LIN {X 0,Y 531.026,Z 365.335,A -85,B 0,C 180,E1 -4215.435,E2 -4215.435} C_VEL
LIN {X 0,Y 531.043,Z 365.34,A -85,B 0,C 180,E1 -4218.549,E2 -4218.549} C_VEL
LIN {X 0,Y 531.061,Z 365.329,A -85,B 0,C 180,E1 -4221.629,E2 -4221.629} C_VEL
LIN {X 0,Y 531.122,Z 365.326,A -85,B 0,C 180,E1 -4224.684,E2 -4224.684} C_VEL
LIN {X 0,Y 531.145,Z 365.319,A -85,B 0,C 180,E1 -4227.724,E2 -4227.724} C_VEL
LIN {X 0,Y 531.157,Z 365.319,A -85,B 0,C 180,E1 -4230.757,E2 -4230.757} C_VEL
LIN {X 0,Y 531.108,Z 365.323,A -85,B 0,C 180,E1 -4233.033,E2 -4233.033} C_VEL
LIN {X 0,Y 531.087,Z 365.332,A -85,B 0,C 180,E1 -4236.076,E2 -4236.076} C_VEL
LIN {X 0,Y 531.056,Z 365.335,A -85,B 0,C 180,E1 -4238.369,E2 -4238.369} C_VEL
LIN {X 0,Y 531.054,Z 365.332,A -85,B 0,C 180,E1 -4241.671,E2 -4241.671} C_VEL
LIN {X 0,Y 531.033,Z 365.332,A -85,B 0,C 180,E1 -4244.955,E2 -4244.955} C_VEL
LIN {X 0,Y 531.018,Z 365.339,A -85,B 0,C 180,E1 -4247.721,E2 -4247.721} C_VEL
LIN {X 0,Y 531.025,Z 365.339,A -85,B 0,C 180,E1 -4250.126,E2 -4250.126} C_VEL
LIN {X 0,Y 530.946,Z 365.344,A -85,B 0,C 180,E1 -4252.572,E2 -4252.572} C_VEL
LIN {X 0,Y 530.994,Z 365.337,A -85,B 0,C 180,E1 -4255.057,E2 -4255.057} C_VEL
LIN {X 0,Y 531.015,Z 365.34,A -85,B 0,C 180,E1 -4257.594,E2 -4257.594} C_VEL
LIN {X 0,Y 530.981,Z 365.339,A -85,B 0,C 180,E1 -4260.646,E2 -4260.646} C_VEL
LIN {X 0,Y 530.988,Z 365.346,A -85,B 0,C 180,E1 -4263.771,E2 -4263.771} C_VEL
LIN {X 0,Y 530.965,Z 365.34,A -85,B 0,C 180,E1 -4266.556,E2 -4266.556} C_VEL
LIN {X 0,Y 530.996,Z 365.341,A -85,B 0,C 180,E1 -4269.855,E2 -4269.855} C_VEL
LIN {X 0,Y 530.978,Z 365.339,A -85,B 0,C 180,E1 -4272.455,E2 -4272.455} C_VEL
LIN {X 0,Y 530.983,Z 365.347,A -85,B 0,C 180,E1 -4275.62,E2 -4275.62} C_VEL
LIN {X 0,Y 531.042,Z 365.474,A -85,B 0,C 180,E1 -4277.77,E2 -4277.77} C_VEL
LIN {X 0,Y 531.558,Z 369.985,A -85,B 0,C 180,E1 -4278.618,E2 -4278.618} C_VEL
LIN {X 0,Y 531.348,Z 387.405,A -85,B 0,C 180,E1 -4281.804,E2 -4281.804} C_VEL
LIN {X 0,Y 531.197,Z 394.529,A -85,B 0,C 180,E1 -4283.118,E2 -4283.118} C_VEL
LIN {X 0,Y 532.782,Z 405.07,A -85,B 0,C 180,E1 -4283.315,E2 -4283.315} C_VEL
LIN {X 0,Y 532.355,Z 500.213,A -85,B 0,C 180,E1 -4284.624,E2 -4284.624} C_VEL
LIN {X 0,Y 532.243,Z 511.094,A -85,B 0,C 180,E1 -4284.875,E2 -4284.875} C_VEL
LIN {X 0,Y 532.076,Z 522.958,A -85,B 0,C 180,E1 -4285.275,E2 -4285.275} C_VEL
LIN {X 0,Y 531.831,Z 535.01,A -85,B 0,C 180,E1 -4285.831,E2 -4285.831} C_VEL
LIN {X 0,Y 531.61,Z 545.985,A -85,B 0,C 180,E1 -4286.499,E2 -4286.499} C_VEL
LIN {X 0,Y 531.342,Z 555.982,A -85,B 0,C 180,E1 -4287.257,E2 -4287.257} C_VEL
LIN {X 0,Y 531.14,Z 564.562,A -85,B 0,C 180,E1 -4288.043,E2 -4288.043} C_VEL
LIN {X 0,Y 530.97,Z 572.57,A -85,B 0,C 180,E1 -4288.921,E2 -4288.921} C_VEL
LIN {X 0,Y 530.813,Z 579.244,A -85,B 0,C 180,E1 -4289.793,E2 -4289.793} C_VEL
LIN {X 0,Y 530.664,Z 584.849,A -85,B 0,C 180,E1 -4290.658,E2 -4290.658} C_VEL
LIN {X 0,Y 530.582,Z 590.653,A -85,B 0,C 180,E1 -4291.736,E2 -4291.736} C_VEL
LIN {X 0,Y 530.512,Z 595.671,A -85,B 0,C 180,E1 -4292.899,E2 -4292.899} C_VEL
LIN {X 0,Y 530.466,Z 600.121,A -85,B 0,C 180,E1 -4294.275,E2 -4294.275} C_VEL
LIN {X 0,Y 530.387,Z 603.167,A -85,B 0,C 180,E1 -4295.746,E2 -4295.746} C_VEL
LIN {X 0,Y 530.394,Z 604.282,A -85,B 0,C 180,E1 -4296.577,E2 -4296.577} C_VEL
LIN {X 0,Y 530.349,Z 604.907,A -85,B 0,C 180,E1 -4297.4,E2 -4297.4} C_VEL
LIN {X 0,Y 530.396,Z 604.976,A -85,B 0,C 180,E1 -4298.222,E2 -4298.222} C_VEL
LIN {X 0,Y 530.35,Z 603.932,A -85,B 0,C 180,E1 -4299.846,E2 -4299.846} C_VEL
LIN {X 0,Y 530.381,Z 602.696,A -85,B 0,C 180,E1 -4300.654,E2 -4300.654} C_VEL
LIN {X 0,Y 530.464,Z 600.013,A -85,B 0,C 180,E1 -4301.859,E2 -4301.859} C_VEL
LIN {X 0,Y 530.485,Z 596.223,A -85,B 0,C 180,E1 -4303.054,E2 -4303.054} C_VEL
LIN {X 0,Y 530.552,Z 591.215,A -85,B 0,C 180,E1 -4304.243,E2 -4304.243} C_VEL
LIN {X 0,Y 530.673,Z 586.337,A -85,B 0,C 180,E1 -4305.185,E2 -4305.185} C_VEL
LIN {X 0,Y 530.795,Z 579.863,A -85,B 0,C 180,E1 -4306.212,E2 -4306.212} C_VEL
LIN {X 0,Y 530.963,Z 572.403,A -85,B 0,C 180,E1 -4307.19,E2 -4307.19} C_VEL
LIN {X 0,Y 531.141,Z 564.201,A -85,B 0,C 180,E1 -4308.085,E2 -4308.085} C_VEL
LIN {X 0,Y 531.385,Z 554.7,A -85,B 0,C 180,E1 -4308.944,E2 -4308.944} C_VEL
LIN {X 0,Y 531.696,Z 542.537,A -85,B 0,C 180,E1 -4309.817,E2 -4309.817} C_VEL
LIN {X 0,Y 531.902,Z 531.205,A -85,B 0,C 180,E1 -4310.445,E2 -4310.445} C_VEL
LIN {X 0,Y 532.087,Z 519.921,A -85,B 0,C 180,E1 -4310.928,E2 -4310.928} C_VEL
LIN {X 0,Y 532.288,Z 507.418,A -85,B 0,C 180,E1 -4311.314,E2 -4311.314} C_VEL
LIN {X 0,Y 532.422,Z 491.23,A -85,B 0,C 180,E1 -4311.603,E2 -4311.603} C_VEL
LIN {X 0,Y 532.675,Z 403.02,A -85,B 0,C 180,E1 -4312.807,E2 -4312.807} C_VEL
LIN {X 0,Y 531.213,Z 394.5,A -85,B 0,C 180,E1 -4312.992,E2 -4312.992} C_VEL
LIN {X 0,Y 531.363,Z 379.959,A -85,B 0,C 180,E1 -4315.638,E2 -4315.638} C_VEL
LIN {X 0,Y 531.455,Z 369.437,A -85,B 0,C 180,E1 -4317.537,E2 -4317.537} C_VEL
LIN {X 0,Y 531.071,Z 365.336,A -85,B 0,C 180,E1 -4318.294,E2 -4318.294} C_VEL
LIN {X 0,Y 531.147,Z 365.326,A -85,B 0,C 180,E1 -4320.758,E2 -4320.758} C_VEL
LIN {X 0,Y 531.101,Z 365.329,A -85,B 0,C 180,E1 -4323.034,E2 -4323.034} C_VEL
LIN {X 0,Y 531.075,Z 365.333,A -85,B 0,C 180,E1 -4326.077,E2 -4326.077} C_VEL
LIN {X 0,Y 531.027,Z 365.335,A -85,B 0,C 180,E1 -4329.138,E2 -4329.138} C_VEL
LIN {X 0,Y 531.031,Z 365.34,A -85,B 0,C 180,E1 -4332.225,E2 -4332.225} C_VEL
LIN {X 0,Y 530.987,Z 365.34,A -85,B 0,C 180,E1 -4335.35,E2 -4335.35} C_VEL
LIN {X 0,Y 531.006,Z 365.341,A -85,B 0,C 180,E1 -4337.723,E2 -4337.723} C_VEL
LIN {X 0,Y 530.998,Z 365.337,A -85,B 0,C 180,E1 -4340.938,E2 -4340.938} C_VEL
LIN {X 0,Y 531.018,Z 365.341,A -85,B 0,C 180,E1 -4344.05,E2 -4344.05} C_VEL
LIN {X 0,Y 531.006,Z 365.336,A -85,B 0,C 180,E1 -4346.744,E2 -4346.744} C_VEL
LIN {X 0,Y 530.991,Z 365.342,A -85,B 0,C 180,E1 -4349.322,E2 -4349.322} C_VEL
LIN {X 0,Y 530.972,Z 365.343,A -85,B 0,C 180,E1 -4352.104,E2 -4352.104} C_VEL
LIN {X 0,Y 530.983,Z 365.34,A -85,B 0,C 180,E1 -4354.855,E2 -4354.855} C_VEL
LIN {X 0,Y 530.959,Z 365.35,A -85,B 0,C 180,E1 -4357.508,E2 -4357.508} C_VEL
LIN {X 0,Y 530.978,Z 365.34,A -85,B 0,C 180,E1 -4360.433,E2 -4360.433} C_VEL
LIN {X 0,Y 530.961,Z 365.347,A -85,B 0,C 180,E1 -4363.495,E2 -4363.495} C_VEL
LIN {X 0,Y 530.958,Z 365.343,A -85,B 0,C 180,E1 -4366.507,E2 -4366.507} C_VEL
LIN {X 0,Y 530.984,Z 365.346,A -85,B 0,C 180,E1 -4368.977,E2 -4368.977} C_VEL
LIN {X 0,Y 530.955,Z 365.345,A -85,B 0,C 180,E1 -4371.531,E2 -4371.531} C_VEL
LIN {X 0,Y 530.979,Z 365.341,A -85,B 0,C 180,E1 -4374.383,E2 -4374.383} C_VEL
LIN {X 0,Y 530.969,Z 365.346,A -85,B 0,C 180,E1 -4377.135,E2 -4377.135} C_VEL
LIN {X 0,Y 530.984,Z 365.34,A -85,B 0,C 180,E1 -4379.805,E2 -4379.805} C_VEL
LIN {X 0,Y 531.016,Z 365.341,A -85,B 0,C 180,E1 -4382.467,E2 -4382.467} C_VEL
LIN {X 0,Y 531.007,Z 365.344,A -85,B 0,C 180,E1 -4384.944,E2 -4384.944} C_VEL
LIN {X 0,Y 531.039,Z 365.539,A -85,B 0,C 180,E1 -4386.001,E2 -4386.001} C_VEL
LIN {X 0,Y 532.353,Z 373.078,A -85,B 0,C 180,E1 -4387.286,E2 -4387.286} C_VEL
LIN {X 0,Y 531.956,Z 390.881,A -85,B 0,C 180,E1 -4390.112,E2 -4390.112} C_VEL
LIN {X 0,Y 531.575,Z 408.654,A -85,B 0,C 180,E1 -4392.893,E2 -4392.893} C_VEL
LIN {X 0,Y 531.338,Z 422.569,A -85,B 0,C 180,E1 -4395.054,E2 -4395.054} C_VEL
LIN {X 0,Y 532.834,Z 432.971,A -85,B 0,C 180,E1 -4395.239,E2 -4395.239} C_VEL
LIN {X 0,Y 532.412,Z 530.394,A -85,B 0,C 180,E1 -4396.572,E2 -4396.572} C_VEL
LIN {X 0,Y 532.216,Z 543.761,A -85,B 0,C 180,E1 -4396.907,E2 -4396.907} C_VEL
LIN {X 0,Y 531.997,Z 555.976,A -85,B 0,C 180,E1 -4397.363,E2 -4397.363} C_VEL
LIN {X 0,Y 531.74,Z 568.122,A -85,B 0,C 180,E1 -4397.976,E2 -4397.976} C_VEL
LIN {X 0,Y 531.507,Z 579.917,A -85,B 0,C 180,E1 -4398.754,E2 -4398.754} C_VEL
LIN {X 0,Y 531.219,Z 590.378,A -85,B 0,C 180,E1 -4399.616,E2 -4399.616} C_VEL
LIN {X 0,Y 531.032,Z 598.931,A -85,B 0,C 180,E1 -4400.479,E2 -4400.479} C_VEL
LIN {X 0,Y 530.885,Z 606.821,A -85,B 0,C 180,E1 -4401.436,E2 -4401.436} C_VEL
LIN {X 0,Y 530.68,Z 614.522,A -85,B 0,C 180,E1 -4402.582,E2 -4402.582} C_VEL
LIN {X 0,Y 530.604,Z 621.622,A -85,B 0,C 180,E1 -4403.918,E2 -4403.918} C_VEL
LIN {X 0,Y 530.459,Z 626.341,A -85,B 0,C 180,E1 -4405.061,E2 -4405.061} C_VEL
LIN {X 0,Y 530.516,Z 629.95,A -85,B 0,C 180,E1 -4406.203,E2 -4406.203} C_VEL
LIN {X 0,Y 530.457,Z 631.806,A -85,B 0,C 180,E1 -4406.963,E2 -4406.963} C_VEL
LIN {X 0,Y 530.41,Z 633.194,A -85,B 0,C 180,E1 -4407.723,E2 -4407.723} C_VEL
LIN {X 0,Y 530.344,Z 634.786,A -85,B 0,C 180,E1 -4409.242,E2 -4409.242} C_VEL
LIN {X 0,Y 530.342,Z 635,A -85,B 0,C 180,E1 -4410.001,E2 -4410.001} C_VEL
LIN {X 0,Y 530.361,Z 634.182,A -85,B 0,C 180,E1 -4411.52,E2 -4411.52} C_VEL
LIN {X 0,Y 530.411,Z 633.194,A -85,B 0,C 180,E1 -4412.279,E2 -4412.279} C_VEL
LIN {X 0,Y 530.457,Z 631.805,A -85,B 0,C 180,E1 -4413.039,E2 -4413.039} C_VEL
LIN {X 0,Y 530.523,Z 628.874,A -85,B 0,C 180,E1 -4414.179,E2 -4414.179} C_VEL
LIN {X 0,Y 530.525,Z 624.9,A -85,B 0,C 180,E1 -4415.322,E2 -4415.322} C_VEL
LIN {X 0,Y 530.6,Z 619.178,A -85,B 0,C 180,E1 -4416.583,E2 -4416.583} C_VEL
LIN {X 0,Y 530.737,Z 612.104,A -85,B 0,C 180,E1 -4417.802,E2 -4417.802} C_VEL
LIN {X 0,Y 530.929,Z 603.811,A -85,B 0,C 180,E1 -4418.949,E2 -4418.949} C_VEL
LIN {X 0,Y 531.123,Z 595.305,A -85,B 0,C 180,E1 -4419.906,E2 -4419.906} C_VEL
LIN {X 0,Y 531.379,Z 584.793,A -85,B 0,C 180,E1 -4420.864,E2 -4420.864} C_VEL
LIN {X 0,Y 531.632,Z 573.998,A -85,B 0,C 180,E1 -4421.658,E2 -4421.658} C_VEL
LIN {X 0,Y 531.895,Z 562.981,A -85,B 0,C 180,E1 -4422.303,E2 -4422.303} C_VEL
LIN {X 0,Y 532.107,Z 551.244,A -85,B 0,C 180,E1 -4422.831,E2 -4422.831} C_VEL
LIN {X 0,Y 532.277,Z 538.628,A -85,B 0,C 180,E1 -4423.239,E2 -4423.239} C_VEL
LIN {X 0,Y 532.477,Z 525.779,A -85,B 0,C 180,E1 -4423.501,E2 -4423.501} C_VEL
LIN {X 0,Y 532.689,Z 431.415,A -85,B 0,C 180,E1 -4424.784,E2 -4424.784} C_VEL
LIN {X 0,Y 531.306,Z 422.381,A -85,B 0,C 180,E1 -4424.964,E2 -4424.964} C_VEL
LIN {X 0,Y 531.733,Z 402.026,A -85,B 0,C 180,E1 -4428.119,E2 -4428.119} C_VEL
LIN {X 0,Y 532.124,Z 381.772,A -85,B 0,C 180,E1 -4431.298,E2 -4431.298} C_VEL
LIN {X 0,Y 532.319,Z 372.885,A -85,B 0,C 180,E1 -4432.718,E2 -4432.718} C_VEL
LIN {X 0,Y 531.008,Z 365.342,A -85,B 0,C 180,E1 -4434.032,E2 -4434.032} C_VEL
LIN {X 0,Y 531.01,Z 365.339,A -85,B 0,C 180,E1 -4436.744,E2 -4436.744} C_VEL
LIN {X 0,Y 530.988,Z 365.348,A -85,B 0,C 180,E1 -4439.323,E2 -4439.323} C_VEL
LIN {X 0,Y 530.972,Z 365.342,A -85,B 0,C 180,E1 -4442.101,E2 -4442.101} C_VEL
LIN {X 0,Y 530.986,Z 365.343,A -85,B 0,C 180,E1 -4444.853,E2 -4444.853} C_VEL
LIN {X 0,Y 530.972,Z 365.346,A -85,B 0,C 180,E1 -4447.508,E2 -4447.508} C_VEL
LIN {X 0,Y 530.987,Z 365.341,A -85,B 0,C 180,E1 -4450.433,E2 -4450.433} C_VEL
LIN {X 0,Y 530.971,Z 365.344,A -85,B 0,C 180,E1 -4453.495,E2 -4453.495} C_VEL
LIN {X 0,Y 530.971,Z 365.344,A -85,B 0,C 180,E1 -4456.506,E2 -4456.506} C_VEL
LIN {X 0,Y 530.986,Z 365.338,A -85,B 0,C 180,E1 -4459.567,E2 -4459.567} C_VEL
LIN {X 0,Y 530.973,Z 365.345,A -85,B 0,C 180,E1 -4462.577,E2 -4462.577} C_VEL
LIN {X 0,Y 530.987,Z 365.339,A -85,B 0,C 180,E1 -4465.31,E2 -4465.31} C_VEL
LIN {X 0,Y 530.972,Z 365.341,A -85,B 0,C 180,E1 -4468.032,E2 -4468.032} C_VEL
LIN {X 0,Y 530.994,Z 365.343,A -85,B 0,C 180,E1 -4470.875,E2 -4470.875} C_VEL
LIN {X 0,Y 531.003,Z 365.335,A -85,B 0,C 180,E1 -4473.256,E2 -4473.256} C_VEL
LIN {X 0,Y 530.965,Z 365.343,A -85,B 0,C 180,E1 -4475.967,E2 -4475.967} C_VEL
LIN {X 0,Y 531.005,Z 365.338,A -85,B 0,C 180,E1 -4479.062,E2 -4479.062} C_VEL
LIN {X 0,Y 531.022,Z 365.338,A -85,B 0,C 180,E1 -4482.278,E2 -4482.278} C_VEL
LIN {X 0,Y 531.025,Z 365.331,A -85,B 0,C 180,E1 -4485.436,E2 -4485.436} C_VEL
LIN {X 0,Y 531.043,Z 365.335,A -85,B 0,C 180,E1 -4488.55,E2 -4488.55} C_VEL
LIN {X 0,Y 531.06,Z 365.331,A -85,B 0,C 180,E1 -4491.63,E2 -4491.63} C_VEL
LIN {X 0,Y 531.126,Z 365.323,A -85,B 0,C 180,E1 -4494.685,E2 -4494.685} C_VEL
LIN {X 0,Y 531.145,Z 365.32,A -85,B 0,C 180,E1 -4497.725,E2 -4497.725} C_VEL
LIN {X 0,Y 531.158,Z 365.317,A -85,B 0,C 180,E1 -4500.758,E2 -4500.758} C_VEL
LIN {X 0,Y 531.11,Z 365.323,A -85,B 0,C 180,E1 -4503.034,E2 -4503.034} C_VEL
LIN {X 0,Y 531.09,Z 365.332,A -85,B 0,C 180,E1 -4506.077,E2 -4506.077} C_VEL
LIN {X 0,Y 531.034,Z 365.333,A -85,B 0,C 180,E1 -4509.138,E2 -4509.138} C_VEL
LIN {X 0,Y 531.047,Z 365.335,A -85,B 0,C 180,E1 -4512.225,E2 -4512.225} C_VEL
LIN {X 0,Y 531.002,Z 365.34,A -85,B 0,C 180,E1 -4515.35,E2 -4515.35} C_VEL
LIN {X 0,Y 530.994,Z 365.339,A -85,B 0,C 180,E1 -4518.521,E2 -4518.521} C_VEL
LIN {X 0,Y 531.006,Z 365.338,A -85,B 0,C 180,E1 -4520.938,E2 -4520.938} C_VEL
LIN {X 0,Y 530.972,Z 365.343,A -85,B 0,C 180,E1 -4524.225,E2 -4524.225} C_VEL
LIN {X 0,Y 531.006,Z 365.338,A -85,B 0,C 180,E1 -4526.744,E2 -4526.744} C_VEL
LIN {X 0,Y 530.987,Z 365.347,A -85,B 0,C 180,E1 -4529.323,E2 -4529.323} C_VEL
LIN {X 0,Y 531.017,Z 365.438,A -85,B 0,C 180,E1 -4531.491,E2 -4531.491} C_VEL
LIN {X 0,Y 531.738,Z 370.239,A -85,B 0,C 180,E1 -4532.452,E2 -4532.452} C_VEL
LIN {X 0,Y 531.385,Z 386.614,A -85,B 0,C 180,E1 -4535.587,E2 -4535.587} C_VEL
LIN {X 0,Y 531.254,Z 394.792,A -85,B 0,C 180,E1 -4537.104,E2 -4537.104} C_VEL
LIN {X 0,Y 532.829,Z 404.238,A -85,B 0,C 180,E1 -4537.289,E2 -4537.289} C_VEL
LIN {X 0,Y 532.733,Z 424.698,A -85,B 0,C 180,E1 -4537.566,E2 -4537.566} C_VEL
LIN {X 0,Y 532.089,Z 430.539,A -85,B 0,C 180,E1 -4537.627,E2 -4537.627} C_VEL
LIN {X 0,Y 526.454,Z 449.535,A -85,B 0,C 180,E1 -4537.733,E2 -4537.733} C_VEL
LIN {X 0,Y 525.731,Z 455.378,A -85,B 0,C 180,E1 -4537.795,E2 -4537.795} C_VEL
LIN {X 0,Y 525.475,Z 502.765,A -85,B 0,C 180,E1 -4538.472,E2 -4538.472} C_VEL
LIN {X 0,Y 525.32,Z 516.428,A -85,B 0,C 180,E1 -4538.838,E2 -4538.838} C_VEL
LIN {X 0,Y 525.063,Z 528.553,A -85,B 0,C 180,E1 -4539.321,E2 -4539.321} C_VEL
LIN {X 0,Y 524.808,Z 540.204,A -85,B 0,C 180,E1 -4539.941,E2 -4539.941} C_VEL
LIN {X 0,Y 524.541,Z 551.45,A -85,B 0,C 180,E1 -4540.71,E2 -4540.71} C_VEL
LIN {X 0,Y 524.204,Z 561.789,A -85,B 0,C 180,E1 -4541.595,E2 -4541.595} C_VEL
LIN {X 0,Y 523.964,Z 571.304,A -85,B 0,C 180,E1 -4542.601,E2 -4542.601} C_VEL
LIN {X 0,Y 523.739,Z 580.071,A -85,B 0,C 180,E1 -4543.753,E2 -4543.753} C_VEL
LIN {X 0,Y 523.569,Z 587.846,A -85,B 0,C 180,E1 -4545.033,E2 -4545.033} C_VEL
LIN {X 0,Y 523.494,Z 593.113,A -85,B 0,C 180,E1 -4546.125,E2 -4546.125} C_VEL
LIN {X 0,Y 523.431,Z 597.338,A -85,B 0,C 180,E1 -4547.224,E2 -4547.224} C_VEL
LIN {X 0,Y 523.379,Z 600.599,A -85,B 0,C 180,E1 -4548.326,E2 -4548.326} C_VEL
LIN {X 0,Y 523.273,Z 603.65,A -85,B 0,C 180,E1 -4549.857,E2 -4549.857} C_VEL
LIN {X 0,Y 523.25,Z 604.987,A -85,B 0,C 180,E1 -4551.172,E2 -4551.172} C_VEL
LIN {X 0,Y 523.236,Z 605.194,A -85,B 0,C 180,E1 -4552.418,E2 -4552.418} C_VEL
LIN {X 0,Y 523.249,Z 604.258,A -85,B 0,C 180,E1 -4553.772,E2 -4553.772} C_VEL
LIN {X 0,Y 523.29,Z 602.309,A -85,B 0,C 180,E1 -4555.011,E2 -4555.011} C_VEL
LIN {X 0,Y 523.404,Z 598.941,A -85,B 0,C 180,E1 -4556.357,E2 -4556.357} C_VEL
LIN {X 0,Y 523.474,Z 593.949,A -85,B 0,C 180,E1 -4557.76,E2 -4557.76} C_VEL
LIN {X 0,Y 523.574,Z 588.89,A -85,B 0,C 180,E1 -4558.852,E2 -4558.852} C_VEL
LIN {X 0,Y 523.748,Z 582.223,A -85,B 0,C 180,E1 -4560.009,E2 -4560.009} C_VEL
LIN {X 0,Y 523.919,Z 574.268,A -85,B 0,C 180,E1 -4561.123,E2 -4561.123} C_VEL
LIN {X 0,Y 524.182,Z 564.373,A -85,B 0,C 180,E1 -4562.24,E2 -4562.24} C_VEL
LIN {X 0,Y 524.447,Z 554.824,A -85,B 0,C 180,E1 -4563.109,E2 -4563.109} C_VEL
LIN {X 0,Y 524.733,Z 544.034,A -85,B 0,C 180,E1 -4563.904,E2 -4563.904} C_VEL
LIN {X 0,Y 525.004,Z 532.385,A -85,B 0,C 180,E1 -4564.582,E2 -4564.582} C_VEL
LIN {X 0,Y 525.233,Z 519.897,A -85,B 0,C 180,E1 -4565.129,E2 -4565.129} C_VEL
LIN {X 0,Y 525.465,Z 506.906,A -85,B 0,C 180,E1 -4565.525,E2 -4565.525} C_VEL
LIN {X 0,Y 525.546,Z 493.531,A -85,B 0,C 180,E1 -4565.771,E2 -4565.771} C_VEL
LIN {X 0,Y 525.814,Z 403.589,A -85,B 0,C 180,E1 -4567.011,E2 -4567.011} C_VEL
LIN {X 0,Y 524.213,Z 394.773,A -85,B 0,C 180,E1 -4567.2,E2 -4567.2} C_VEL
LIN {X 0,Y 524.624,Z 377.867,A -85,B 0,C 180,E1 -4570.432,E2 -4570.432} C_VEL
LIN {X 0,Y 524.728,Z 371.323,A -85,B 0,C 180,E1 -4571.694,E2 -4571.694} C_VEL
LIN {X 0,Y 524.02,Z 366.215,A -85,B 0,C 180,E1 -4572.758,E2 -4572.758} C_VEL
LIN {X 0,Y 523.984,Z 366.214,A -85,B 0,C 180,E1 -4575.235,E2 -4575.235} C_VEL
LIN {X 0,Y 524.019,Z 366.213,A -85,B 0,C 180,E1 -4578.393,E2 -4578.393} C_VEL
LIN {X 0,Y 524.009,Z 366.207,A -85,B 0,C 180,E1 -4581.515,E2 -4581.515} C_VEL
LIN {X 0,Y 524.082,Z 366.204,A -85,B 0,C 180,E1 -4584.613,E2 -4584.613} C_VEL
LIN {X 0,Y 524.117,Z 366.194,A -85,B 0,C 180,E1 -4587.694,E2 -4587.694} C_VEL
LIN {X 0,Y 524.128,Z 366.195,A -85,B 0,C 180,E1 -4590.767,E2 -4590.767} C_VEL
LIN {X 0,Y 524.075,Z 366.199,A -85,B 0,C 180,E1 -4593.074,E2 -4593.074} C_VEL
LIN {X 0,Y 524.049,Z 366.21,A -85,B 0,C 180,E1 -4596.158,E2 -4596.158} C_VEL
LIN {X 0,Y 524.004,Z 366.212,A -85,B 0,C 180,E1 -4598.483,E2 -4598.483} C_VEL
LIN {X 0,Y 524.005,Z 366.211,A -85,B 0,C 180,E1 -4601.738,E2 -4601.738} C_VEL
LIN {X 0,Y 523.995,Z 366.209,A -85,B 0,C 180,E1 -4605.051,E2 -4605.051} C_VEL
LIN {X 0,Y 523.965,Z 366.222,A -85,B 0,C 180,E1 -4607.968,E2 -4607.968} C_VEL
LIN {X 0,Y 523.972,Z 366.214,A -85,B 0,C 180,E1 -4610.409,E2 -4610.409} C_VEL
LIN {X 0,Y 523.911,Z 366.219,A -85,B 0,C 180,E1 -4612.892,E2 -4612.892} C_VEL
LIN {X 0,Y 523.983,Z 366.216,A -85,B 0,C 180,E1 -4616.019,E2 -4616.019} C_VEL
LIN {X 0,Y 523.942,Z 366.215,A -85,B 0,C 180,E1 -4618.873,E2 -4618.873} C_VEL
LIN {X 0,Y 523.931,Z 366.223,A -85,B 0,C 180,E1 -4621.542,E2 -4621.542} C_VEL
LIN {X 0,Y 523.942,Z 366.217,A -85,B 0,C 180,E1 -4624.288,E2 -4624.288} C_VEL
LIN {X 0,Y 523.908,Z 366.222,A -85,B 0,C 180,E1 -4627.13,E2 -4627.13} C_VEL
LIN {X 0,Y 523.964,Z 366.214,A -85,B 0,C 180,E1 -4630.133,E2 -4630.133} C_VEL
LIN {X 0,Y 523.92,Z 366.222,A -85,B 0,C 180,E1 -4633.165,E2 -4633.165} C_VEL
LIN {X 0,Y 523.936,Z 366.223,A -85,B 0,C 180,E1 -4635.771,E2 -4635.771} C_VEL
LIN {X 0,Y 523.99,Z 366.422,A -85,B 0,C 180,E1 -4637.688,E2 -4637.688} C_VEL
LIN {X 0,Y 524.555,Z 371.275,A -85,B 0,C 180,E1 -4638.613,E2 -4638.613} C_VEL
LIN {X 0,Y 524.33,Z 388.067,A -85,B 0,C 180,E1 -4641.703,E2 -4641.703} C_VEL
LIN {X 0,Y 524.241,Z 394.6,A -85,B 0,C 180,E1 -4642.912,E2 -4642.912} C_VEL
LIN {X 0,Y 525.918,Z 405.618,A -85,B 0,C 180,E1 -4643.127,E2 -4643.127} C_VEL
LIN {X 0,Y 525.442,Z 501.337,A -85,B 0,C 180,E1 -4644.472,E2 -4644.472} C_VEL
LIN {X 0,Y 525.283,Z 514.4,A -85,B 0,C 180,E1 -4644.799,E2 -4644.799} C_VEL
LIN {X 0,Y 525.056,Z 528.066,A -85,B 0,C 180,E1 -4645.328,E2 -4645.328} C_VEL
LIN {X 0,Y 524.802,Z 538.765,A -85,B 0,C 180,E1 -4645.888,E2 -4645.888} C_VEL
LIN {X 0,Y 524.579,Z 548.161,A -85,B 0,C 180,E1 -4646.499,E2 -4646.499} C_VEL
LIN {X 0,Y 524.309,Z 557.464,A -85,B 0,C 180,E1 -4647.234,E2 -4647.234} C_VEL
LIN {X 0,Y 524.089,Z 566.794,A -85,B 0,C 180,E1 -4648.128,E2 -4648.128} C_VEL
LIN {X 0,Y 523.888,Z 575.574,A -85,B 0,C 180,E1 -4649.153,E2 -4649.153} C_VEL
LIN {X 0,Y 523.656,Z 583.023,A -85,B 0,C 180,E1 -4650.226,E2 -4650.226} C_VEL
LIN {X 0,Y 523.55,Z 589.192,A -85,B 0,C 180,E1 -4651.321,E2 -4651.321} C_VEL
LIN {X 0,Y 523.431,Z 594.1,A -85,B 0,C 180,E1 -4652.392,E2 -4652.392} C_VEL
LIN {X 0,Y 523.414,Z 598.737,A -85,B 0,C 180,E1 -4653.698,E2 -4653.698} C_VEL
LIN {X 0,Y 523.367,Z 601.052,A -85,B 0,C 180,E1 -4654.551,E2 -4654.551} C_VEL
LIN {X 0,Y 523.299,Z 602.874,A -85,B 0,C 180,E1 -4655.396,E2 -4655.396} C_VEL
LIN {X 0,Y 523.294,Z 604.144,A -85,B 0,C 180,E1 -4656.24,E2 -4656.24} C_VEL
LIN {X 0,Y 523.271,Z 604.87,A -85,B 0,C 180,E1 -4657.077,E2 -4657.077} C_VEL
LIN {X 0,Y 523.276,Z 605.175,A -85,B 0,C 180,E1 -4657.926,E2 -4657.926} C_VEL
LIN {X 0,Y 523.267,Z 605.071,A -85,B 0,C 180,E1 -4658.738,E2 -4658.738} C_VEL
LIN {X 0,Y 523.295,Z 603.829,A -85,B 0,C 180,E1 -4660.067,E2 -4660.067} C_VEL
LIN {X 0,Y 523.297,Z 601.853,A -85,B 0,C 180,E1 -4661.196,E2 -4661.196} C_VEL
LIN {X 0,Y 523.388,Z 598.631,A -85,B 0,C 180,E1 -4662.431,E2 -4662.431} C_VEL
LIN {X 0,Y 523.42,Z 594.421,A -85,B 0,C 180,E1 -4663.622,E2 -4663.622} C_VEL
LIN {X 0,Y 523.545,Z 588.969,A -85,B 0,C 180,E1 -4664.82,E2 -4664.82} C_VEL
LIN {X 0,Y 523.73,Z 582.052,A -85,B 0,C 180,E1 -4666.022,E2 -4666.022} C_VEL
LIN {X 0,Y 523.854,Z 574.998,A -85,B 0,C 180,E1 -4667.014,E2 -4667.014} C_VEL
LIN {X 0,Y 524.092,Z 566.674,A -85,B 0,C 180,E1 -4667.977,E2 -4667.977} C_VEL
LIN {X 0,Y 524.311,Z 558.211,A -85,B 0,C 180,E1 -4668.792,E2 -4668.792} C_VEL
LIN {X 0,Y 524.512,Z 549.697,A -85,B 0,C 180,E1 -4669.481,E2 -4669.481} C_VEL
LIN {X 0,Y 524.824,Z 539.297,A -85,B 0,C 180,E1 -4670.169,E2 -4670.169} C_VEL
LIN {X 0,Y 525.062,Z 528.134,A -85,B 0,C 180,E1 -4670.757,E2 -4670.757} C_VEL
LIN {X 0,Y 525.28,Z 514.971,A -85,B 0,C 180,E1 -4671.27,E2 -4671.27} C_VEL
LIN {X 0,Y 525.462,Z 502.139,A -85,B 0,C 180,E1 -4671.598,E2 -4671.598} C_VEL
LIN {X 0,Y 525.743,Z 435.252,A -85,B 0,C 180,E1 -4672.551,E2 -4672.551} C_VEL
LIN {X 0,Y 525.914,Z 404.47,A -85,B 0,C 180,E1 -4672.98,E2 -4672.98} C_VEL
LIN {X 0,Y 524.202,Z 394.667,A -85,B 0,C 180,E1 -4673.19,E2 -4673.19} C_VEL
LIN {X 0,Y 524.46,Z 377.377,A -85,B 0,C 180,E1 -4676.35,E2 -4676.35} C_VEL
LIN {X 0,Y 524.376,Z 368.838,A -85,B 0,C 180,E1 -4677.888,E2 -4677.888} C_VEL
LIN {X 0,Y 524.012,Z 366.216,A -85,B 0,C 180,E1 -4678.415,E2 -4678.415} C_VEL
LIN {X 0,Y 524.117,Z 366.202,A -85,B 0,C 180,E1 -4680.768,E2 -4680.768} C_VEL
LIN {X 0,Y 524.067,Z 366.205,A -85,B 0,C 180,E1 -4683.075,E2 -4683.075} C_VEL
LIN {X 0,Y 524.037,Z 366.211,A -85,B 0,C 180,E1 -4686.159,E2 -4686.159} C_VEL
LIN {X 0,Y 523.994,Z 366.211,A -85,B 0,C 180,E1 -4689.262,E2 -4689.262} C_VEL
LIN {X 0,Y 524.013,Z 366.211,A -85,B 0,C 180,E1 -4691.751,E2 -4691.751} C_VEL
LIN {X 0,Y 523.981,Z 366.212,A -85,B 0,C 180,E1 -4695.053,E2 -4695.053} C_VEL
LIN {X 0,Y 523.954,Z 366.223,A -85,B 0,C 180,E1 -4697.969,E2 -4697.969} C_VEL
LIN {X 0,Y 523.964,Z 366.217,A -85,B 0,C 180,E1 -4700.41,E2 -4700.41} C_VEL
LIN {X 0,Y 523.947,Z 366.215,A -85,B 0,C 180,E1 -4702.892,E2 -4702.892} C_VEL
LIN {X 0,Y 523.954,Z 366.218,A -85,B 0,C 180,E1 -4705.419,E2 -4705.419} C_VEL
LIN {X 0,Y 523.962,Z 366.219,A -85,B 0,C 180,E1 -4707.999,E2 -4707.999} C_VEL
LIN {X 0,Y 523.944,Z 366.217,A -85,B 0,C 180,E1 -4710.857,E2 -4710.857} C_VEL
LIN {X 0,Y 523.954,Z 366.221,A -85,B 0,C 180,E1 -4713.736,E2 -4713.736} C_VEL
LIN {X 0,Y 523.914,Z 366.22,A -85,B 0,C 180,E1 -4716.405,E2 -4716.405} C_VEL
LIN {X 0,Y 523.919,Z 366.223,A -85,B 0,C 180,E1 -4719.085,E2 -4719.085} C_VEL
LIN {X 0,Y 523.951,Z 366.215,A -85,B 0,C 180,E1 -4722.119,E2 -4722.119} C_VEL
LIN {X 0,Y 523.949,Z 366.222,A -85,B 0,C 180,E1 -4725.31,E2 -4725.31} C_VEL
LIN {X 0,Y 523.956,Z 366.217,A -85,B 0,C 180,E1 -4728.69,E2 -4728.69} C_VEL
LIN {X 0,Y 523.913,Z 366.22,A -85,B 0,C 180,E1 -4731.9,E2 -4731.9} C_VEL
LIN {X 0,Y 523.935,Z 366.225,A -85,B 0,C 180,E1 -4734.91,E2 -4734.91} C_VEL
LIN {X 0,Y 523.94,Z 366.217,A -85,B 0,C 180,E1 -4737.679,E2 -4737.679} C_VEL
LIN {X 0,Y 523.968,Z 366.221,A -85,B 0,C 180,E1 -4740.674,E2 -4740.674} C_VEL
LIN {X 0,Y 523.976,Z 366.214,A -85,B 0,C 180,E1 -4743.73,E2 -4743.73} C_VEL
LIN {X 0,Y 523.968,Z 366.245,A -85,B 0,C 180,E1 -4745.796,E2 -4745.796} C_VEL
LIN {X 0,Y 525.406,Z 374.198,A -85,B 0,C 180,E1 -4747.177,E2 -4747.177} C_VEL
LIN {X 0,Y 524.989,Z 391.985,A -85,B 0,C 180,E1 -4750.041,E2 -4750.041} C_VEL
LIN {X 0,Y 524.52,Z 411.012,A -85,B 0,C 180,E1 -4753.058,E2 -4753.058} C_VEL
LIN {X 0,Y 524.322,Z 422.578,A -85,B 0,C 180,E1 -4754.852,E2 -4754.852} C_VEL
LIN {X 0,Y 525.975,Z 433.876,A -85,B 0,C 180,E1 -4755.059,E2 -4755.059} C_VEL
LIN {X 0,Y 525.488,Z 531.193,A -85,B 0,C 180,E1 -4756.416,E2 -4756.416} C_VEL
LIN {X 0,Y 525.249,Z 544.984,A -85,B 0,C 180,E1 -4756.779,E2 -4756.779} C_VEL
LIN {X 0,Y 525.027,Z 557.869,A -85,B 0,C 180,E1 -4757.29,E2 -4757.29} C_VEL
LIN {X 0,Y 524.687,Z 570.261,A -85,B 0,C 180,E1 -4757.96,E2 -4757.96} C_VEL
LIN {X 0,Y 524.482,Z 580.972,A -85,B 0,C 180,E1 -4758.7,E2 -4758.7} C_VEL
LIN {X 0,Y 524.171,Z 591.196,A -85,B 0,C 180,E1 -4759.573,E2 -4759.573} C_VEL
LIN {X 0,Y 523.952,Z 600.389,A -85,B 0,C 180,E1 -4760.544,E2 -4760.544} C_VEL
LIN {X 0,Y 523.732,Z 609.344,A -85,B 0,C 180,E1 -4761.707,E2 -4761.707} C_VEL
LIN {X 0,Y 523.582,Z 616.55,A -85,B 0,C 180,E1 -4762.869,E2 -4762.869} C_VEL
LIN {X 0,Y 523.523,Z 623.112,A -85,B 0,C 180,E1 -4764.223,E2 -4764.223} C_VEL
LIN {X 0,Y 523.36,Z 627.448,A -85,B 0,C 180,E1 -4765.38,E2 -4765.38} C_VEL
LIN {X 0,Y 523.443,Z 629.747,A -85,B 0,C 180,E1 -4766.152,E2 -4766.152} C_VEL
LIN {X 0,Y 523.367,Z 631.607,A -85,B 0,C 180,E1 -4766.922,E2 -4766.922} C_VEL
LIN {X 0,Y 523.334,Z 633.001,A -85,B 0,C 180,E1 -4767.692,E2 -4767.692} C_VEL
LIN {X 0,Y 523.25,Z 634.602,A -85,B 0,C 180,E1 -4769.231,E2 -4769.231} C_VEL
LIN {X 0,Y 523.246,Z 634.817,A -85,B 0,C 180,E1 -4770.001,E2 -4770.001} C_VEL
LIN {X 0,Y 523.275,Z 633.993,A -85,B 0,C 180,E1 -4771.54,E2 -4771.54} C_VEL
LIN {X 0,Y 523.334,Z 632.999,A -85,B 0,C 180,E1 -4772.31,E2 -4772.31} C_VEL
LIN {X 0,Y 523.368,Z 631.602,A -85,B 0,C 180,E1 -4773.08,E2 -4773.08} C_VEL
LIN {X 0,Y 523.425,Z 628.665,A -85,B 0,C 180,E1 -4774.236,E2 -4774.236} C_VEL
LIN {X 0,Y 523.464,Z 624.687,A -85,B 0,C 180,E1 -4775.394,E2 -4775.394} C_VEL
LIN {X 0,Y 523.522,Z 619.434,A -85,B 0,C 180,E1 -4776.58,E2 -4776.58} C_VEL
LIN {X 0,Y 523.655,Z 613.115,A -85,B 0,C 180,E1 -4777.714,E2 -4777.714} C_VEL
LIN {X 0,Y 523.836,Z 605.07,A -85,B 0,C 180,E1 -4778.876,E2 -4778.876} C_VEL
LIN {X 0,Y 524.06,Z 596.868,A -85,B 0,C 180,E1 -4779.846,E2 -4779.846} C_VEL
LIN {X 0,Y 524.338,Z 586.863,A -85,B 0,C 180,E1 -4780.817,E2 -4780.817} C_VEL
LIN {X 0,Y 524.608,Z 575.581,A -85,B 0,C 180,E1 -4781.689,E2 -4781.689} C_VEL
LIN {X 0,Y 524.873,Z 564.47,A -85,B 0,C 180,E1 -4782.372,E2 -4782.372} C_VEL
LIN {X 0,Y 525.152,Z 552.175,A -85,B 0,C 180,E1 -4782.954,E2 -4782.954} C_VEL
LIN {X 0,Y 525.349,Z 539.186,A -85,B 0,C 180,E1 -4783.392,E2 -4783.392} C_VEL
LIN {X 0,Y 525.558,Z 526.835,A -85,B 0,C 180,E1 -4783.658,E2 -4783.658} C_VEL
LIN {X 0,Y 525.78,Z 431.837,A -85,B 0,C 180,E1 -4784.974,E2 -4784.974} C_VEL
LIN {X 0,Y 524.284,Z 422.16,A -85,B 0,C 180,E1 -4785.169,E2 -4785.169} C_VEL
LIN {X 0,Y 524.744,Z 402.218,A -85,B 0,C 180,E1 -4788.306,E2 -4788.306} C_VEL
LIN {X 0,Y 525.182,Z 382.86,A -85,B 0,C 180,E1 -4791.388,E2 -4791.388} C_VEL
LIN {X 0,Y 525.35,Z 373.989,A -85,B 0,C 180,E1 -4792.828,E2 -4792.828} C_VEL
LIN {X 0,Y 523.967,Z 366.219,A -85,B 0,C 180,E1 -4794.204,E2 -4794.204} C_VEL
LIN {X 0,Y 523.959,Z 366.222,A -85,B 0,C 180,E1 -4797.133,E2 -4797.133} C_VEL
LIN {X 0,Y 523.948,Z 366.22,A -85,B 0,C 180,E1 -4799.756,E2 -4799.756} C_VEL
LIN {X 0,Y 523.939,Z 366.218,A -85,B 0,C 180,E1 -4802.45,E2 -4802.45} C_VEL
LIN {X 0,Y 523.93,Z 366.226,A -85,B 0,C 180,E1 -4805.227,E2 -4805.227} C_VEL
LIN {X 0,Y 523.922,Z 366.22,A -85,B 0,C 180,E1 -4808.102,E2 -4808.102} C_VEL
LIN {X 0,Y 523.945,Z 366.226,A -85,B 0,C 180,E1 -4811.093,E2 -4811.093} C_VEL
LIN {X 0,Y 523.947,Z 366.217,A -85,B 0,C 180,E1 -4814.228,E2 -4814.228} C_VEL
LIN {X 0,Y 523.927,Z 366.226,A -85,B 0,C 180,E1 -4816.834,E2 -4816.834} C_VEL
LIN {X 0,Y 523.943,Z 366.214,A -85,B 0,C 180,E1 -4819.871,E2 -4819.871} C_VEL
LIN {X 0,Y 523.912,Z 366.226,A -85,B 0,C 180,E1 -4822.868,E2 -4822.868} C_VEL
LIN {X 0,Y 523.938,Z 366.215,A -85,B 0,C 180,E1 -4825.71,E2 -4825.71} C_VEL
LIN {X 0,Y 523.926,Z 366.223,A -85,B 0,C 180,E1 -4828.456,E2 -4828.456} C_VEL
LIN {X 0,Y 523.94,Z 366.219,A -85,B 0,C 180,E1 -4831.125,E2 -4831.125} C_VEL
LIN {X 0,Y 523.989,Z 366.209,A -85,B 0,C 180,E1 -4833.981,E2 -4833.981} C_VEL
LIN {X 0,Y 523.917,Z 366.218,A -85,B 0,C 180,E1 -4837.107,E2 -4837.107} C_VEL
LIN {X 0,Y 523.985,Z 366.212,A -85,B 0,C 180,E1 -4839.866,E2 -4839.866} C_VEL
LIN {X 0,Y 523.972,Z 366.216,A -85,B 0,C 180,E1 -4842.837,E2 -4842.837} C_VEL
LIN {X 0,Y 523.983,Z 366.208,A -85,B 0,C 180,E1 -4845.236,E2 -4845.236} C_VEL
LIN {X 0,Y 524.018,Z 366.212,A -85,B 0,C 180,E1 -4848.394,E2 -4848.394} C_VEL
LIN {X 0,Y 524.009,Z 366.208,A -85,B 0,C 180,E1 -4851.516,E2 -4851.516} C_VEL
LIN {X 0,Y 524.088,Z 366.201,A -85,B 0,C 180,E1 -4854.614,E2 -4854.614} C_VEL
LIN {X 0,Y 524.117,Z 366.195,A -85,B 0,C 180,E1 -4857.695,E2 -4857.695} C_VEL
LIN {X 0,Y 524.128,Z 366.192,A -85,B 0,C 180,E1 -4860.768,E2 -4860.768} C_VEL
LIN {X 0,Y 524.077,Z 366.199,A -85,B 0,C 180,E1 -4863.075,E2 -4863.075} C_VEL
LIN {X 0,Y 524.052,Z 366.207,A -85,B 0,C 180,E1 -4866.159,E2 -4866.159} C_VEL
LIN {X 0,Y 524.002,Z 366.21,A -85,B 0,C 180,E1 -4869.262,E2 -4869.262} C_VEL
LIN {X 0,Y 524.009,Z 366.216,A -85,B 0,C 180,E1 -4871.739,E2 -4871.739} C_VEL
LIN {X 0,Y 523.999,Z 366.21,A -85,B 0,C 180,E1 -4875.052,E2 -4875.052} C_VEL
LIN {X 0,Y 523.97,Z 366.219,A -85,B 0,C 180,E1 -4877.969,E2 -4877.969} C_VEL
LIN {X 0,Y 523.978,Z 366.213,A -85,B 0,C 180,E1 -4880.41,E2 -4880.41} C_VEL
LIN {X 0,Y 523.917,Z 366.221,A -85,B 0,C 180,E1 -4882.893,E2 -4882.893} C_VEL
LIN {X 0,Y 523.99,Z 366.214,A -85,B 0,C 180,E1 -4886.02,E2 -4886.02} C_VEL
LIN {X 0,Y 523.944,Z 366.219,A -85,B 0,C 180,E1 -4888.875,E2 -4888.875} C_VEL
LIN {X 0,Y 523.956,Z 366.262,A -85,B 0,C 180,E1 -4891.332,E2 -4891.332} C_VEL
LIN {X 0,Y 524.782,Z 371.864,A -85,B 0,C 180,E1 -4892.465,E2 -4892.465} C_VEL
LIN {X 0,Y 524.39,Z 388.403,A -85,B 0,C 180,E1 -4895.662,E2 -4895.662} C_VEL
LIN {X 0,Y 524.236,Z 394.928,A -85,B 0,C 180,E1 -4896.903,E2 -4896.903} C_VEL
LIN {X 0,Y 525.972,Z 404.789,A -85,B 0,C 180,E1 -4897.099,E2 -4897.099} C_VEL
LIN {X 0,Y 525.731,Z 455.378,A -85,B 0,C 180,E1 -4897.795,E2 -4897.795} C_VEL
LIN {X 0,Y 524.992,Z 461.222,A -85,B 0,C 180,E1 -4897.856,E2 -4897.856} C_VEL
LIN {X 0,Y 519.301,Z 480.202,A -85,B 0,C 180,E1 -4897.966,E2 -4897.966} C_VEL
LIN {X 0,Y 518.714,Z 486.041,A -85,B 0,C 180,E1 -4898.032,E2 -4898.032} C_VEL
LIN {X 0,Y 518.588,Z 504.633,A -85,B 0,C 180,E1 -4898.328,E2 -4898.328} C_VEL
LIN {X 0,Y 518.411,Z 516.016,A -85,B 0,C 180,E1 -4898.643,E2 -4898.643} C_VEL
LIN {X 0,Y 518.202,Z 527.597,A -85,B 0,C 180,E1 -4899.098,E2 -4899.098} C_VEL
LIN {X 0,Y 517.899,Z 539.983,A -85,B 0,C 180,E1 -4899.755,E2 -4899.755} C_VEL
LIN {X 0,Y 517.57,Z 551.567,A -85,B 0,C 180,E1 -4900.553,E2 -4900.553} C_VEL
LIN {X 0,Y 517.225,Z 561.667,A -85,B 0,C 180,E1 -4901.424,E2 -4901.424} C_VEL
LIN {X 0,Y 517.011,Z 570.46,A -85,B 0,C 180,E1 -4902.353,E2 -4902.353} C_VEL
LIN {X 0,Y 516.766,Z 578.254,A -85,B 0,C 180,E1 -4903.348,E2 -4903.348} C_VEL
LIN {X 0,Y 516.589,Z 585.323,A -85,B 0,C 180,E1 -4904.448,E2 -4904.448} C_VEL
LIN {X 0,Y 516.437,Z 592.202,A -85,B 0,C 180,E1 -4905.795,E2 -4905.795} C_VEL
LIN {X 0,Y 516.353,Z 597.379,A -85,B 0,C 180,E1 -4907.113,E2 -4907.113} C_VEL
LIN {X 0,Y 516.286,Z 601.292,A -85,B 0,C 180,E1 -4908.478,E2 -4908.478} C_VEL
LIN {X 0,Y 516.186,Z 603.644,A -85,B 0,C 180,E1 -4909.681,E2 -4909.681} C_VEL
LIN {X 0,Y 516.166,Z 605.223,A -85,B 0,C 180,E1 -4911.22,E2 -4911.22} C_VEL
LIN {X 0,Y 516.133,Z 605.437,A -85,B 0,C 180,E1 -4912.211,E2 -4912.211} C_VEL
LIN {X 0,Y 516.156,Z 604.803,A -85,B 0,C 180,E1 -4913.451,E2 -4913.451} C_VEL
LIN {X 0,Y 516.183,Z 603.005,A -85,B 0,C 180,E1 -4914.778,E2 -4914.778} C_VEL
LIN {X 0,Y 516.306,Z 599.937,A -85,B 0,C 180,E1 -4916.134,E2 -4916.134} C_VEL
LIN {X 0,Y 516.368,Z 595.295,A -85,B 0,C 180,E1 -4917.549,E2 -4917.549} C_VEL
LIN {X 0,Y 516.501,Z 589.482,A -85,B 0,C 180,E1 -4918.864,E2 -4918.864} C_VEL
LIN {X 0,Y 516.702,Z 582.013,A -85,B 0,C 180,E1 -4920.18,E2 -4920.18} C_VEL
LIN {X 0,Y 516.915,Z 573.53,A -85,B 0,C 180,E1 -4921.362,E2 -4921.362} C_VEL
LIN {X 0,Y 517.198,Z 563.51,A -85,B 0,C 180,E1 -4922.482,E2 -4922.482} C_VEL
LIN {X 0,Y 517.526,Z 553.569,A -85,B 0,C 180,E1 -4923.375,E2 -4923.375} C_VEL
LIN {X 0,Y 517.837,Z 542.621,A -85,B 0,C 180,E1 -4924.168,E2 -4924.168} C_VEL
LIN {X 0,Y 518.102,Z 531.336,A -85,B 0,C 180,E1 -4924.811,E2 -4924.811} C_VEL
LIN {X 0,Y 518.349,Z 519.369,A -85,B 0,C 180,E1 -4925.329,E2 -4925.329} C_VEL
LIN {X 0,Y 518.569,Z 506.038,A -85,B 0,C 180,E1 -4925.731,E2 -4925.731} C_VEL
LIN {X 0,Y 518.689,Z 491.047,A -85,B 0,C 180,E1 -4925.99,E2 -4925.99} C_VEL
LIN {X 0,Y 519.011,Z 404.718,A -85,B 0,C 180,E1 -4927.199,E2 -4927.199} C_VEL
LIN {X 0,Y 517.229,Z 394.996,A -85,B 0,C 180,E1 -4927.403,E2 -4927.403} C_VEL
LIN {X 0,Y 517.658,Z 378.615,A -85,B 0,C 180,E1 -4930.571,E2 -4930.571} C_VEL
LIN {X 0,Y 517.658,Z 371.194,A -85,B 0,C 180,E1 -4932.028,E2 -4932.028} C_VEL
LIN {X 0,Y 516.967,Z 367.093,A -85,B 0,C 180,E1 -4932.902,E2 -4932.902} C_VEL
LIN {X 0,Y 516.902,Z 367.095,A -85,B 0,C 180,E1 -4935.833,E2 -4935.833} C_VEL
LIN {X 0,Y 516.972,Z 367.089,A -85,B 0,C 180,E1 -4938.233,E2 -4938.233} C_VEL
LIN {X 0,Y 516.974,Z 367.083,A -85,B 0,C 180,E1 -4941.399,E2 -4941.399} C_VEL
LIN {X 0,Y 517.029,Z 367.084,A -85,B 0,C 180,E1 -4944.539,E2 -4944.539} C_VEL
LIN {X 0,Y 517.089,Z 367.07,A -85,B 0,C 180,E1 -4947.662,E2 -4947.662} C_VEL
LIN {X 0,Y 517.098,Z 367.071,A -85,B 0,C 180,E1 -4950.778,E2 -4950.778} C_VEL
LIN {X 0,Y 517.016,Z 367.078,A -85,B 0,C 180,E1 -4953.116,E2 -4953.116} C_VEL
LIN {X 0,Y 517.013,Z 367.087,A -85,B 0,C 180,E1 -4956.242,E2 -4956.242} C_VEL
LIN {X 0,Y 516.948,Z 367.087,A -85,B 0,C 180,E1 -4959.388,E2 -4959.388} C_VEL
LIN {X 0,Y 516.955,Z 367.09,A -85,B 0,C 180,E1 -4961.806,E2 -4961.806} C_VEL
LIN {X 0,Y 516.946,Z 367.087,A -85,B 0,C 180,E1 -4965.145,E2 -4965.145} C_VEL
LIN {X 0,Y 516.926,Z 367.095,A -85,B 0,C 180,E1 -4968.221,E2 -4968.221} C_VEL
LIN {X 0,Y 516.912,Z 367.092,A -85,B 0,C 180,E1 -4970.7,E2 -4970.7} C_VEL
LIN {X 0,Y 516.887,Z 367.1,A -85,B 0,C 180,E1 -4974.072,E2 -4974.072} C_VEL
LIN {X 0,Y 516.925,Z 367.09,A -85,B 0,C 180,E1 -4976.656,E2 -4976.656} C_VEL
LIN {X 0,Y 516.918,Z 367.096,A -85,B 0,C 180,E1 -4979.524,E2 -4979.524} C_VEL
LIN {X 0,Y 516.898,Z 367.093,A -85,B 0,C 180,E1 -4982.543,E2 -4982.543} C_VEL
LIN {X 0,Y 516.881,Z 367.099,A -85,B 0,C 180,E1 -4985.331,E2 -4985.331} C_VEL
LIN {X 0,Y 516.878,Z 367.099,A -85,B 0,C 180,E1 -4987.942,E2 -4987.942} C_VEL
LIN {X 0,Y 516.89,Z 367.094,A -85,B 0,C 180,E1 -4990.739,E2 -4990.739} C_VEL
LIN {X 0,Y 516.877,Z 367.101,A -85,B 0,C 180,E1 -4993.892,E2 -4993.892} C_VEL
LIN {X 0,Y 516.877,Z 367.099,A -85,B 0,C 180,E1 -4996.106,E2 -4996.106} C_VEL
LIN {X 0,Y 516.973,Z 367.283,A -85,B 0,C 180,E1 -4997.589,E2 -4997.589} C_VEL
LIN {X 0,Y 517.58,Z 372.472,A -85,B 0,C 180,E1 -4998.576,E2 -4998.576} C_VEL
LIN {X 0,Y 517.305,Z 389.308,A -85,B 0,C 180,E1 -5001.699,E2 -5001.699} C_VEL
LIN {X 0,Y 517.254,Z 394.693,A -85,B 0,C 180,E1 -5002.695,E2 -5002.695} C_VEL
LIN {X 0,Y 519.077,Z 406.705,A -85,B 0,C 180,E1 -5002.942,E2 -5002.942} C_VEL
LIN {X 0,Y 518.532,Z 501.961,A -85,B 0,C 180,E1 -5004.307,E2 -5004.307} C_VEL
LIN {X 0,Y 518.359,Z 514.754,A -85,B 0,C 180,E1 -5004.636,E2 -5004.636} C_VEL
LIN {X 0,Y 518.106,Z 527.903,A -85,B 0,C 180,E1 -5005.151,E2 -5005.151} C_VEL
LIN {X 0,Y 517.861,Z 538.467,A -85,B 0,C 180,E1 -5005.705,E2 -5005.705} C_VEL
LIN {X 0,Y 517.599,Z 549.054,A -85,B 0,C 180,E1 -5006.406,E2 -5006.406} C_VEL
LIN {X 0,Y 517.307,Z 558.691,A -85,B 0,C 180,E1 -5007.19,E2 -5007.19} C_VEL
LIN {X 0,Y 517.008,Z 568.928,A -85,B 0,C 180,E1 -5008.213,E2 -5008.213} C_VEL
LIN {X 0,Y 516.797,Z 577.895,A -85,B 0,C 180,E1 -5009.338,E2 -5009.338} C_VEL
LIN {X 0,Y 516.563,Z 584.958,A -85,B 0,C 180,E1 -5010.427,E2 -5010.427} C_VEL
LIN {X 0,Y 516.434,Z 590.922,A -85,B 0,C 180,E1 -5011.555,E2 -5011.555} C_VEL
LIN {X 0,Y 516.352,Z 596.433,A -85,B 0,C 180,E1 -5012.873,E2 -5012.873} C_VEL
LIN {X 0,Y 516.288,Z 600.474,A -85,B 0,C 180,E1 -5014.176,E2 -5014.176} C_VEL
LIN {X 0,Y 516.222,Z 602.442,A -85,B 0,C 180,E1 -5015.036,E2 -5015.036} C_VEL
LIN {X 0,Y 516.231,Z 603.859,A -85,B 0,C 180,E1 -5015.894,E2 -5015.894} C_VEL
LIN {X 0,Y 516.172,Z 604.827,A -85,B 0,C 180,E1 -5016.743,E2 -5016.743} C_VEL
LIN {X 0,Y 516.182,Z 605.374,A -85,B 0,C 180,E1 -5017.792,E2 -5017.792} C_VEL
LIN {X 0,Y 516.171,Z 605.366,A -85,B 0,C 180,E1 -5018.431,E2 -5018.431} C_VEL
LIN {X 0,Y 516.213,Z 604.235,A -85,B 0,C 180,E1 -5019.947,E2 -5019.947} C_VEL
LIN {X 0,Y 516.196,Z 602.714,A -85,B 0,C 180,E1 -5020.928,E2 -5020.928} C_VEL
LIN {X 0,Y 516.302,Z 599.304,A -85,B 0,C 180,E1 -5022.331,E2 -5022.331} C_VEL
LIN {X 0,Y 516.32,Z 595.802,A -85,B 0,C 180,E1 -5023.39,E2 -5023.39} C_VEL
LIN {X 0,Y 516.464,Z 590.583,A -85,B 0,C 180,E1 -5024.612,E2 -5024.612} C_VEL
LIN {X 0,Y 516.618,Z 584.046,A -85,B 0,C 180,E1 -5025.826,E2 -5025.826} C_VEL
LIN {X 0,Y 516.816,Z 575.898,A -85,B 0,C 180,E1 -5027.034,E2 -5027.034} C_VEL
LIN {X 0,Y 517.082,Z 566.712,A -85,B 0,C 180,E1 -5028.118,E2 -5028.118} C_VEL
LIN {X 0,Y 517.324,Z 558.303,A -85,B 0,C 180,E1 -5028.937,E2 -5028.937} C_VEL
LIN {X 0,Y 517.604,Z 548.395,A -85,B 0,C 180,E1 -5029.734,E2 -5029.734} C_VEL
LIN {X 0,Y 517.914,Z 537.661,A -85,B 0,C 180,E1 -5030.431,E2 -5030.431} C_VEL
LIN {X 0,Y 518.171,Z 524.771,A -85,B 0,C 180,E1 -5031.076,E2 -5031.076} C_VEL
LIN {X 0,Y 518.379,Z 511.747,A -85,B 0,C 180,E1 -5031.539,E2 -5031.539} C_VEL
LIN {X 0,Y 518.538,Z 499.132,A -85,B 0,C 180,E1 -5031.83,E2 -5031.83} C_VEL
LIN {X 0,Y 519.003,Z 404.747,A -85,B 0,C 180,E1 -5033.18,E2 -5033.18} C_VEL
LIN {X 0,Y 517.202,Z 394.847,A -85,B 0,C 180,E1 -5033.397,E2 -5033.397} C_VEL
LIN {X 0,Y 517.466,Z 377.873,A -85,B 0,C 180,E1 -5036.496,E2 -5036.496} C_VEL
LIN {X 0,Y 517.312,Z 369.318,A -85,B 0,C 180,E1 -5038.054,E2 -5038.054} C_VEL
LIN {X 0,Y 516.968,Z 367.093,A -85,B 0,C 180,E1 -5038.491,E2 -5038.491} C_VEL
LIN {X 0,Y 517.086,Z 367.078,A -85,B 0,C 180,E1 -5040.779,E2 -5040.779} C_VEL
LIN {X 0,Y 517.008,Z 367.084,A -85,B 0,C 180,E1 -5043.117,E2 -5043.117} C_VEL
LIN {X 0,Y 517.001,Z 367.089,A -85,B 0,C 180,E1 -5046.243,E2 -5046.243} C_VEL
LIN {X 0,Y 516.948,Z 367.088,A -85,B 0,C 180,E1 -5049.389,E2 -5049.389} C_VEL
LIN {X 0,Y 516.972,Z 367.089,A -85,B 0,C 180,E1 -5051.824,E2 -5051.824} C_VEL
LIN {X 0,Y 516.933,Z 367.09,A -85,B 0,C 180,E1 -5055.147,E2 -5055.147} C_VEL
LIN {X 0,Y 516.916,Z 367.098,A -85,B 0,C 180,E1 -5058.223,E2 -5058.223} C_VEL
LIN {X 0,Y 516.907,Z 367.093,A -85,B 0,C 180,E1 -5060.702,E2 -5060.702} C_VEL
LIN {X 0,Y 516.895,Z 367.095,A -85,B 0,C 180,E1 -5063.222,E2 -5063.222} C_VEL
LIN {X 0,Y 516.938,Z 367.092,A -85,B 0,C 180,E1 -5066.198,E2 -5066.198} C_VEL
LIN {X 0,Y 516.927,Z 367.094,A -85,B 0,C 180,E1 -5069.304,E2 -5069.304} C_VEL
LIN {X 0,Y 516.893,Z 367.095,A -85,B 0,C 180,E1 -5072.545,E2 -5072.545} C_VEL
LIN {X 0,Y 516.875,Z 367.103,A -85,B 0,C 180,E1 -5075.333,E2 -5075.333} C_VEL
LIN {X 0,Y 516.874,Z 367.099,A -85,B 0,C 180,E1 -5077.944,E2 -5077.944} C_VEL
LIN {X 0,Y 516.878,Z 367.098,A -85,B 0,C 180,E1 -5080.742,E2 -5080.742} C_VEL
LIN {X 0,Y 516.898,Z 367.096,A -85,B 0,C 180,E1 -5082.83,E2 -5082.83} C_VEL
LIN {X 0,Y 516.916,Z 367.097,A -85,B 0,C 180,E1 -5085.011,E2 -5085.011} C_VEL
LIN {X 0,Y 516.911,Z 367.093,A -85,B 0,C 180,E1 -5088.399,E2 -5088.399} C_VEL
LIN {X 0,Y 516.879,Z 367.102,A -85,B 0,C 180,E1 -5091.286,E2 -5091.286} C_VEL
LIN {X 0,Y 516.887,Z 367.096,A -85,B 0,C 180,E1 -5094.223,E2 -5094.223} C_VEL
LIN {X 0,Y 516.894,Z 367.1,A -85,B 0,C 180,E1 -5097.055,E2 -5097.055} C_VEL
LIN {X 0,Y 516.9,Z 367.095,A -85,B 0,C 180,E1 -5099.798,E2 -5099.798} C_VEL
LIN {X 0,Y 516.929,Z 367.096,A -85,B 0,C 180,E1 -5102.469,E2 -5102.469} C_VEL
LIN {X 0,Y 516.906,Z 367.099,A -85,B 0,C 180,E1 -5105.396,E2 -5105.396} C_VEL
LIN {X 0,Y 516.933,Z 367.207,A -85,B 0,C 180,E1 -5105.631,E2 -5105.631} C_VEL
LIN {X 0,Y 518.472,Z 376.049,A -85,B 0,C 180,E1 -5107.184,E2 -5107.184} C_VEL
LIN {X 0,Y 518.018,Z 393.139,A -85,B 0,C 180,E1 -5109.976,E2 -5109.976} C_VEL
LIN {X 0,Y 517.551,Z 410.82,A -85,B 0,C 180,E1 -5112.823,E2 -5112.823} C_VEL
LIN {X 0,Y 517.293,Z 422.155,A -85,B 0,C 180,E1 -5114.633,E2 -5114.633} C_VEL
LIN {X 0,Y 519.103,Z 434.58,A -85,B 0,C 180,E1 -5114.87,E2 -5114.87} C_VEL
LIN {X 0,Y 518.594,Z 530.843,A -85,B 0,C 180,E1 -5116.232,E2 -5116.232} C_VEL
LIN {X 0,Y 518.333,Z 544.681,A -85,B 0,C 180,E1 -5116.6,E2 -5116.6} C_VEL
LIN {X 0,Y 518.067,Z 557.602,A -85,B 0,C 180,E1 -5117.117,E2 -5117.117} C_VEL
LIN {X 0,Y 517.744,Z 569.802,A -85,B 0,C 180,E1 -5117.783,E2 -5117.783} C_VEL
LIN {X 0,Y 517.5,Z 580.73,A -85,B 0,C 180,E1 -5118.545,E2 -5118.545} C_VEL
LIN {X 0,Y 517.19,Z 590.966,A -85,B 0,C 180,E1 -5119.43,E2 -5119.43} C_VEL
LIN {X 0,Y 516.928,Z 600.167,A -85,B 0,C 180,E1 -5120.414,E2 -5120.414} C_VEL
LIN {X 0,Y 516.667,Z 609.126,A -85,B 0,C 180,E1 -5121.593,E2 -5121.593} C_VEL
LIN {X 0,Y 516.509,Z 616.339,A -85,B 0,C 180,E1 -5122.771,E2 -5122.771} C_VEL
LIN {X 0,Y 516.434,Z 622.905,A -85,B 0,C 180,E1 -5124.143,E2 -5124.143} C_VEL
LIN {X 0,Y 516.271,Z 627.244,A -85,B 0,C 180,E1 -5125.316,E2 -5125.316} C_VEL
LIN {X 0,Y 516.352,Z 629.545,A -85,B 0,C 180,E1 -5126.099,E2 -5126.099} C_VEL
LIN {X 0,Y 516.282,Z 631.406,A -85,B 0,C 180,E1 -5126.88,E2 -5126.88} C_VEL
LIN {X 0,Y 516.26,Z 632.802,A -85,B 0,C 180,E1 -5127.66,E2 -5127.66} C_VEL
LIN {X 0,Y 516.16,Z 634.402,A -85,B 0,C 180,E1 -5129.221,E2 -5129.221} C_VEL
LIN {X 0,Y 516.154,Z 634.617,A -85,B 0,C 180,E1 -5130.001,E2 -5130.001} C_VEL
LIN {X 0,Y 516.192,Z 633.791,A -85,B 0,C 180,E1 -5131.561,E2 -5131.561} C_VEL
LIN {X 0,Y 516.261,Z 632.796,A -85,B 0,C 180,E1 -5132.342,E2 -5132.342} C_VEL
LIN {X 0,Y 516.283,Z 631.396,A -85,B 0,C 180,E1 -5133.122,E2 -5133.122} C_VEL
LIN {X 0,Y 516.313,Z 628.455,A -85,B 0,C 180,E1 -5134.294,E2 -5134.294} C_VEL
LIN {X 0,Y 516.381,Z 624.473,A -85,B 0,C 180,E1 -5135.468,E2 -5135.468} C_VEL
LIN {X 0,Y 516.477,Z 618.577,A -85,B 0,C 180,E1 -5136.794,E2 -5136.794} C_VEL
LIN {X 0,Y 516.608,Z 611.65,A -85,B 0,C 180,E1 -5138.017,E2 -5138.017} C_VEL
LIN {X 0,Y 516.827,Z 603.339,A -85,B 0,C 180,E1 -5139.195,E2 -5139.195} C_VEL
LIN {X 0,Y 517.044,Z 594.813,A -85,B 0,C 180,E1 -5140.179,E2 -5140.179} C_VEL
LIN {X 0,Y 517.377,Z 584.28,A -85,B 0,C 180,E1 -5141.162,E2 -5141.162} C_VEL
LIN {X 0,Y 517.676,Z 573.069,A -85,B 0,C 180,E1 -5142.004,E2 -5142.004} C_VEL
LIN {X 0,Y 517.98,Z 562.41,A -85,B 0,C 180,E1 -5142.639,E2 -5142.639} C_VEL
LIN {X 0,Y 518.242,Z 550.608,A -85,B 0,C 180,E1 -5143.18,E2 -5143.18} C_VEL
LIN {X 0,Y 518.473,Z 536.998,A -85,B 0,C 180,E1 -5143.623,E2 -5143.623} C_VEL
LIN {X 0,Y 518.68,Z 523.231,A -85,B 0,C 180,E1 -5143.892,E2 -5143.892} C_VEL
LIN {X 0,Y 518.991,Z 433.001,A -85,B 0,C 180,E1 -5145.154,E2 -5145.154} C_VEL
LIN {X 0,Y 517.282,Z 421.989,A -85,B 0,C 180,E1 -5145.371,E2 -5145.371} C_VEL
LIN {X 0,Y 517.757,Z 401.739,A -85,B 0,C 180,E1 -5148.603,E2 -5148.603} C_VEL
LIN {X 0,Y 518.244,Z 383.965,A -85,B 0,C 180,E1 -5151.479,E2 -5151.479} C_VEL
LIN {X 0,Y 518.42,Z 375.222,A -85,B 0,C 180,E1 -5152.918,E2 -5152.918} C_VEL
LIN {X 0,Y 516.93,Z 367.095,A -85,B 0,C 180,E1 -5154.368,E2 -5154.368} C_VEL
LIN {X 0,Y 516.932,Z 367.092,A -85,B 0,C 180,E1 -5156.658,E2 -5156.658} C_VEL
LIN {X 0,Y 516.917,Z 367.1,A -85,B 0,C 180,E1 -5159.524,E2 -5159.524} C_VEL
LIN {X 0,Y 516.901,Z 367.096,A -85,B 0,C 180,E1 -5162.544,E2 -5162.544} C_VEL
LIN {X 0,Y 516.876,Z 367.104,A -85,B 0,C 180,E1 -5165.331,E2 -5165.331} C_VEL
LIN {X 0,Y 516.887,Z 367.097,A -85,B 0,C 180,E1 -5167.944,E2 -5167.944} C_VEL
LIN {X 0,Y 516.889,Z 367.1,A -85,B 0,C 180,E1 -5170.742,E2 -5170.742} C_VEL
LIN {X 0,Y 516.889,Z 367.102,A -85,B 0,C 180,E1 -5172.832,E2 -5172.832} C_VEL
LIN {X 0,Y 516.929,Z 367.098,A -85,B 0,C 180,E1 -5175.01,E2 -5175.01} C_VEL
LIN {X 0,Y 516.919,Z 367.093,A -85,B 0,C 180,E1 -5178.399,E2 -5178.399} C_VEL
LIN {X 0,Y 516.885,Z 367.098,A -85,B 0,C 180,E1 -5181.284,E2 -5181.284} C_VEL
LIN {X 0,Y 516.876,Z 367.098,A -85,B 0,C 180,E1 -5184.22,E2 -5184.22} C_VEL
LIN {X 0,Y 516.9,Z 367.098,A -85,B 0,C 180,E1 -5187.053,E2 -5187.053} C_VEL
LIN {X 0,Y 516.897,Z 367.091,A -85,B 0,C 180,E1 -5189.797,E2 -5189.797} C_VEL
LIN {X 0,Y 516.929,Z 367.096,A -85,B 0,C 180,E1 -5192.467,E2 -5192.467} C_VEL
LIN {X 0,Y 516.881,Z 367.098,A -85,B 0,C 180,E1 -5195.07,E2 -5195.07} C_VEL
LIN {X 0,Y 516.874,Z 367.094,A -85,B 0,C 180,E1 -5197.622,E2 -5197.622} C_VEL
LIN {X 0,Y 516.937,Z 367.093,A -85,B 0,C 180,E1 -5200.13,E2 -5200.13} C_VEL
LIN {X 0,Y 516.927,Z 367.096,A -85,B 0,C 180,E1 -5202.596,E2 -5202.596} C_VEL
LIN {X 0,Y 516.948,Z 367.085,A -85,B 0,C 180,E1 -5205.03,E2 -5205.03} C_VEL
LIN {X 0,Y 516.972,Z 367.092,A -85,B 0,C 180,E1 -5208.234,E2 -5208.234} C_VEL
LIN {X 0,Y 516.973,Z 367.084,A -85,B 0,C 180,E1 -5211.4,E2 -5211.4} C_VEL
LIN {X 0,Y 517.016,Z 367.079,A -85,B 0,C 180,E1 -5213.757,E2 -5213.757} C_VEL
LIN {X 0,Y 517.09,Z 367.07,A -85,B 0,C 180,E1 -5217.663,E2 -5217.663} C_VEL
LIN {X 0,Y 517.098,Z 367.068,A -85,B 0,C 180,E1 -5220.779,E2 -5220.779} C_VEL
LIN {X 0,Y 517.018,Z 367.078,A -85,B 0,C 180,E1 -5223.117,E2 -5223.117} C_VEL
LIN {X 0,Y 517.017,Z 367.082,A -85,B 0,C 180,E1 -5226.243,E2 -5226.243} C_VEL
LIN {X 0,Y 516.957,Z 367.089,A -85,B 0,C 180,E1 -5229.389,E2 -5229.389} C_VEL
LIN {X 0,Y 516.958,Z 367.093,A -85,B 0,C 180,E1 -5231.807,E2 -5231.807} C_VEL
LIN {X 0,Y 516.951,Z 367.089,A -85,B 0,C 180,E1 -5235.146,E2 -5235.146} C_VEL
LIN {X 0,Y 516.93,Z 367.093,A -85,B 0,C 180,E1 -5238.222,E2 -5238.222} C_VEL
LIN {X 0,Y 516.919,Z 367.092,A -85,B 0,C 180,E1 -5240.701,E2 -5240.701} C_VEL
LIN {X 0,Y 516.898,Z 367.098,A -85,B 0,C 180,E1 -5244.073,E2 -5244.073} C_VEL
LIN {X 0,Y 516.93,Z 367.092,A -85,B 0,C 180,E1 -5246.658,E2 -5246.658} C_VEL
LIN {X 0,Y 516.917,Z 367.099,A -85,B 0,C 180,E1 -5249.524,E2 -5249.524} C_VEL
LIN {X 0,Y 516.906,Z 367.224,A -85,B 0,C 180,E1 -5251.194,E2 -5251.194} C_VEL
LIN {X 0,Y 517.811,Z 372.706,A -85,B 0,C 180,E1 -5252.324,E2 -5252.324} C_VEL
LIN {X 0,Y 517.42,Z 388.523,A -85,B 0,C 180,E1 -5255.415,E2 -5255.415} C_VEL
LIN {X 0,Y 517.273,Z 395.149,A -85,B 0,C 180,E1 -5256.694,E2 -5256.694} C_VEL
LIN {X 0,Y 519.106,Z 405.265,A -85,B 0,C 180,E1 -5256.901,E2 -5256.901} C_VEL
LIN {X 0,Y 518.714,Z 486.041,A -85,B 0,C 180,E1 -5258.032,E2 -5258.032} C_VEL
LIN {X 0,Y 518.08,Z 491.886,A -85,B 0,C 180,E1 -5258.094,E2 -5258.094} C_VEL
LIN {X 0,Y 515.142,Z 501.357,A -85,B 0,C 180,E1 -5258.164,E2 -5258.164} C_VEL
LIN {X 0,Y 512.197,Z 510.727,A -85,B 0,C 180,E1 -5258.309,E2 -5258.309} C_VEL
LIN {X 0,Y 511.511,Z 516.407,A -85,B 0,C 180,E1 -5258.47,E2 -5258.47} C_VEL
LIN {X 0,Y 511.27,Z 528.62,A -85,B 0,C 180,E1 -5258.962,E2 -5258.962} C_VEL
LIN {X 0,Y 510.955,Z 540.701,A -85,B 0,C 180,E1 -5259.622,E2 -5259.622} C_VEL
LIN {X 0,Y 510.609,Z 552.098,A -85,B 0,C 180,E1 -5260.423,E2 -5260.423} C_VEL
LIN {X 0,Y 510.197,Z 563.024,A -85,B 0,C 180,E1 -5261.392,E2 -5261.392} C_VEL
LIN {X 0,Y 509.895,Z 572.835,A -85,B 0,C 180,E1 -5262.484,E2 -5262.484} C_VEL
LIN {X 0,Y 509.669,Z 580.881,A -85,B 0,C 180,E1 -5263.588,E2 -5263.588} C_VEL
LIN {X 0,Y 509.489,Z 587.536,A -85,B 0,C 180,E1 -5264.709,E2 -5264.709} C_VEL
LIN {X 0,Y 509.354,Z 594.107,A -85,B 0,C 180,E1 -5266.111,E2 -5266.111} C_VEL
LIN {X 0,Y 509.236,Z 598.852,A -85,B 0,C 180,E1 -5267.448,E2 -5267.448} C_VEL
LIN {X 0,Y 509.187,Z 601.667,A -85,B 0,C 180,E1 -5268.507,E2 -5268.507} C_VEL
LIN {X 0,Y 509.113,Z 603.697,A -85,B 0,C 180,E1 -5269.547,E2 -5269.547} C_VEL
LIN {X 0,Y 509.085,Z 605.022,A -85,B 0,C 180,E1 -5270.632,E2 -5270.632} C_VEL
LIN {X 0,Y 509.067,Z 605.641,A -85,B 0,C 180,E1 -5271.899,E2 -5271.899} C_VEL
LIN {X 0,Y 509.056,Z 605.228,A -85,B 0,C 180,E1 -5273.202,E2 -5273.202} C_VEL
LIN {X 0,Y 509.095,Z 603.65,A -85,B 0,C 180,E1 -5274.562,E2 -5274.562} C_VEL
LIN {X 0,Y 509.191,Z 600.872,A -85,B 0,C 180,E1 -5275.908,E2 -5275.908} C_VEL
LIN {X 0,Y 509.253,Z 596.544,A -85,B 0,C 180,E1 -5277.335,E2 -5277.335} C_VEL
LIN {X 0,Y 509.397,Z 592.375,A -85,B 0,C 180,E1 -5278.38,E2 -5278.38} C_VEL
LIN {X 0,Y 509.565,Z 585.324,A -85,B 0,C 180,E1 -5279.773,E2 -5279.773} C_VEL
LIN {X 0,Y 509.763,Z 577.968,A -85,B 0,C 180,E1 -5280.922,E2 -5280.922} C_VEL
LIN {X 0,Y 510.025,Z 568.947,A -85,B 0,C 180,E1 -5282.061,E2 -5282.061} C_VEL
LIN {X 0,Y 510.389,Z 558.543,A -85,B 0,C 180,E1 -5283.117,E2 -5283.117} C_VEL
LIN {X 0,Y 510.733,Z 547.872,A -85,B 0,C 180,E1 -5283.983,E2 -5283.983} C_VEL
LIN {X 0,Y 511.052,Z 535.618,A -85,B 0,C 180,E1 -5284.765,E2 -5284.765} C_VEL
LIN {X 0,Y 511.322,Z 523.865,A -85,B 0,C 180,E1 -5285.338,E2 -5285.338} C_VEL
LIN {X 0,Y 511.599,Z 510.759,A -85,B 0,C 180,E1 -5285.796,E2 -5285.796} C_VEL
LIN {X 0,Y 511.752,Z 498.332,A -85,B 0,C 180,E1 -5286.073,E2 -5286.073} C_VEL
LIN {X 0,Y 512.132,Z 405.238,A -85,B 0,C 180,E1 -5287.402,E2 -5287.402} C_VEL
LIN {X 0,Y 510.251,Z 395.203,A -85,B 0,C 180,E1 -5287.615,E2 -5287.615} C_VEL
LIN {X 0,Y 510.677,Z 379.37,A -85,B 0,C 180,E1 -5290.713,E2 -5290.713} C_VEL
LIN {X 0,Y 510.731,Z 372.756,A -85,B 0,C 180,E1 -5292.027,E2 -5292.027} C_VEL
LIN {X 0,Y 509.907,Z 367.972,A -85,B 0,C 180,E1 -5293.046,E2 -5293.046} C_VEL
LIN {X 0,Y 509.87,Z 367.971,A -85,B 0,C 180,E1 -5295.633,E2 -5295.633} C_VEL
LIN {X 0,Y 509.919,Z 367.967,A -85,B 0,C 180,E1 -5298.874,E2 -5298.874} C_VEL
LIN {X 0,Y 509.957,Z 367.961,A -85,B 0,C 180,E1 -5302.078,E2 -5302.078} C_VEL
LIN {X 0,Y 509.979,Z 367.964,A -85,B 0,C 180,E1 -5304.463,E2 -5304.463} C_VEL
LIN {X 0,Y 510.06,Z 367.945,A -85,B 0,C 180,E1 -5307.63,E2 -5307.63} C_VEL
LIN {X 0,Y 510.068,Z 367.946,A -85,B 0,C 180,E1 -5310.788,E2 -5310.788} C_VEL
LIN {X 0,Y 509.958,Z 367.957,A -85,B 0,C 180,E1 -5313.159,E2 -5313.159} C_VEL
LIN {X 0,Y 509.982,Z 367.962,A -85,B 0,C 180,E1 -5316.328,E2 -5316.328} C_VEL
LIN {X 0,Y 509.914,Z 367.965,A -85,B 0,C 180,E1 -5318.719,E2 -5318.719} C_VEL
LIN {X 0,Y 509.907,Z 367.97,A -85,B 0,C 180,E1 -5321.93,E2 -5321.93} C_VEL
LIN {X 0,Y 509.895,Z 367.965,A -85,B 0,C 180,E1 -5325.241,E2 -5325.241} C_VEL
LIN {X 0,Y 509.89,Z 367.975,A -85,B 0,C 180,E1 -5328,E2 -5328} C_VEL
LIN {X 0,Y 509.85,Z 367.971,A -85,B 0,C 180,E1 -5331,E2 -5331} C_VEL
LIN {X 0,Y 509.823,Z 367.978,A -85,B 0,C 180,E1 -5333.562,E2 -5333.562} C_VEL
LIN {X 0,Y 509.911,Z 367.965,A -85,B 0,C 180,E1 -5336.377,E2 -5336.377} C_VEL
LIN {X 0,Y 509.88,Z 367.967,A -85,B 0,C 180,E1 -5338.843,E2 -5338.843} C_VEL
LIN {X 0,Y 509.825,Z 367.981,A -85,B 0,C 180,E1 -5341.588,E2 -5341.588} C_VEL
LIN {X 0,Y 509.851,Z 367.971,A -85,B 0,C 180,E1 -5344.412,E2 -5344.412} C_VEL
LIN {X 0,Y 509.816,Z 367.98,A -85,B 0,C 180,E1 -5347.339,E2 -5347.339} C_VEL
LIN {X 0,Y 509.853,Z 367.971,A -85,B 0,C 180,E1 -5350.379,E2 -5350.379} C_VEL
LIN {X 0,Y 509.835,Z 367.976,A -85,B 0,C 180,E1 -5353.063,E2 -5353.063} C_VEL
LIN {X 0,Y 509.826,Z 367.981,A -85,B 0,C 180,E1 -5355.791,E2 -5355.791} C_VEL
LIN {X 0,Y 509.89,Z 367.989,A -85,B 0,C 180,E1 -5357.449,E2 -5357.449} C_VEL
LIN {X 0,Y 510.599,Z 374.267,A -85,B 0,C 180,E1 -5358.648,E2 -5358.648} C_VEL
LIN {X 0,Y 510.278,Z 390.697,A -85,B 0,C 180,E1 -5361.723,E2 -5361.723} C_VEL
LIN {X 0,Y 510.257,Z 394.883,A -85,B 0,C 180,E1 -5362.495,E2 -5362.495} C_VEL
LIN {X 0,Y 512.231,Z 407.152,A -85,B 0,C 180,E1 -5362.741,E2 -5362.741} C_VEL
LIN {X 0,Y 511.635,Z 502.507,A -85,B 0,C 180,E1 -5364.137,E2 -5364.137} C_VEL
LIN {X 0,Y 511.421,Z 515.916,A -85,B 0,C 180,E1 -5364.495,E2 -5364.495} C_VEL
LIN {X 0,Y 511.142,Z 529.574,A -85,B 0,C 180,E1 -5365.057,E2 -5365.057} C_VEL
LIN {X 0,Y 510.865,Z 540.571,A -85,B 0,C 180,E1 -5365.664,E2 -5365.664} C_VEL
LIN {X 0,Y 510.527,Z 552.075,A -85,B 0,C 180,E1 -5366.47,E2 -5366.47} C_VEL
LIN {X 0,Y 510.245,Z 561.872,A -85,B 0,C 180,E1 -5367.33,E2 -5367.33} C_VEL
LIN {X 0,Y 509.975,Z 569.968,A -85,B 0,C 180,E1 -5368.188,E2 -5368.188} C_VEL
LIN {X 0,Y 509.722,Z 578.761,A -85,B 0,C 180,E1 -5369.326,E2 -5369.326} C_VEL
LIN {X 0,Y 509.489,Z 586.333,A -85,B 0,C 180,E1 -5370.537,E2 -5370.537} C_VEL
LIN {X 0,Y 509.367,Z 591.593,A -85,B 0,C 180,E1 -5371.574,E2 -5371.574} C_VEL
LIN {X 0,Y 509.27,Z 596.968,A -85,B 0,C 180,E1 -5372.909,E2 -5372.909} C_VEL
LIN {X 0,Y 509.197,Z 600.909,A -85,B 0,C 180,E1 -5374.229,E2 -5374.229} C_VEL
LIN {X 0,Y 509.118,Z 603.736,A -85,B 0,C 180,E1 -5375.652,E2 -5375.652} C_VEL
LIN {X 0,Y 509.094,Z 604.739,A -85,B 0,C 180,E1 -5376.4,E2 -5376.4} C_VEL
LIN {X 0,Y 509.096,Z 605.549,A -85,B 0,C 180,E1 -5377.653,E2 -5377.653} C_VEL
LIN {X 0,Y 509.064,Z 605.326,A -85,B 0,C 180,E1 -5378.964,E2 -5378.964} C_VEL
LIN {X 0,Y 509.117,Z 604.612,A -85,B 0,C 180,E1 -5379.829,E2 -5379.829} C_VEL
LIN {X 0,Y 509.118,Z 603.444,A -85,B 0,C 180,E1 -5380.652,E2 -5380.652} C_VEL
LIN {X 0,Y 509.214,Z 599.969,A -85,B 0,C 180,E1 -5382.23,E2 -5382.23} C_VEL
LIN {X 0,Y 509.254,Z 595.587,A -85,B 0,C 180,E1 -5383.566,E2 -5383.566} C_VEL
LIN {X 0,Y 509.432,Z 589.587,A -85,B 0,C 180,E1 -5384.945,E2 -5384.945} C_VEL
LIN {X 0,Y 509.623,Z 582.343,A -85,B 0,C 180,E1 -5386.238,E2 -5386.238} C_VEL
LIN {X 0,Y 509.812,Z 575.25,A -85,B 0,C 180,E1 -5387.257,E2 -5387.257} C_VEL
LIN {X 0,Y 510.083,Z 565.959,A -85,B 0,C 180,E1 -5388.346,E2 -5388.346} C_VEL
LIN {X 0,Y 510.395,Z 556.11,A -85,B 0,C 180,E1 -5389.287,E2 -5389.287} C_VEL
LIN {X 0,Y 510.708,Z 545.682,A -85,B 0,C 180,E1 -5390.095,E2 -5390.095} C_VEL
LIN {X 0,Y 511.028,Z 534.087,A -85,B 0,C 180,E1 -5390.8,E2 -5390.8} C_VEL
LIN {X 0,Y 511.28,Z 521.766,A -85,B 0,C 180,E1 -5391.373,E2 -5391.373} C_VEL
LIN {X 0,Y 511.505,Z 508.947,A -85,B 0,C 180,E1 -5391.796,E2 -5391.796} C_VEL
LIN {X 0,Y 511.676,Z 494.342,A -85,B 0,C 180,E1 -5392.085,E2 -5392.085} C_VEL
LIN {X 0,Y 512.152,Z 405.505,A -85,B 0,C 180,E1 -5393.376,E2 -5393.376} C_VEL
LIN {X 0,Y 510.247,Z 395.047,A -85,B 0,C 180,E1 -5393.599,E2 -5393.599} C_VEL
LIN {X 0,Y 510.506,Z 377.314,A -85,B 0,C 180,E1 -5396.843,E2 -5396.843} C_VEL
LIN {X 0,Y 510.26,Z 369.821,A -85,B 0,C 180,E1 -5398.224,E2 -5398.224} C_VEL
LIN {X 0,Y 509.942,Z 367.969,A -85,B 0,C 180,E1 -5398.593,E2 -5398.593} C_VEL
LIN {X 0,Y 510.056,Z 367.953,A -85,B 0,C 180,E1 -5400.789,E2 -5400.789} C_VEL
LIN {X 0,Y 509.95,Z 367.964,A -85,B 0,C 180,E1 -5403.16,E2 -5403.16} C_VEL
LIN {X 0,Y 509.968,Z 367.965,A -85,B 0,C 180,E1 -5406.33,E2 -5406.33} C_VEL
LIN {X 0,Y 509.909,Z 367.969,A -85,B 0,C 180,E1 -5408.72,E2 -5408.72} C_VEL
LIN {X 0,Y 509.94,Z 367.966,A -85,B 0,C 180,E1 -5411.931,E2 -5411.931} C_VEL
LIN {X 0,Y 509.882,Z 367.969,A -85,B 0,C 180,E1 -5415.242,E2 -5415.242} C_VEL
LIN {X 0,Y 509.878,Z 367.976,A -85,B 0,C 180,E1 -5418.002,E2 -5418.002} C_VEL
LIN {X 0,Y 509.851,Z 367.972,A -85,B 0,C 180,E1 -5421.002,E2 -5421.002} C_VEL
LIN {X 0,Y 509.855,Z 367.975,A -85,B 0,C 180,E1 -5423.562,E2 -5423.562} C_VEL
LIN {X 0,Y 509.906,Z 367.967,A -85,B 0,C 180,E1 -5426.38,E2 -5426.38} C_VEL
LIN {X 0,Y 509.876,Z 367.969,A -85,B 0,C 180,E1 -5428.844,E2 -5428.844} C_VEL
LIN {X 0,Y 509.819,Z 367.983,A -85,B 0,C 180,E1 -5431.59,E2 -5431.59} C_VEL
LIN {X 0,Y 509.846,Z 367.973,A -85,B 0,C 180,E1 -5434.414,E2 -5434.414} C_VEL
LIN {X 0,Y 509.811,Z 367.983,A -85,B 0,C 180,E1 -5437.341,E2 -5437.341} C_VEL
LIN {X 0,Y 509.831,Z 367.974,A -85,B 0,C 180,E1 -5440.383,E2 -5440.383} C_VEL
LIN {X 0,Y 509.834,Z 367.979,A -85,B 0,C 180,E1 -5443.065,E2 -5443.065} C_VEL
LIN {X 0,Y 509.824,Z 367.976,A -85,B 0,C 180,E1 -5445.793,E2 -5445.793} C_VEL
LIN {X 0,Y 509.853,Z 367.973,A -85,B 0,C 180,E1 -5448.576,E2 -5448.576} C_VEL
LIN {X 0,Y 509.847,Z 367.973,A -85,B 0,C 180,E1 -5451.787,E2 -5451.787} C_VEL
LIN {X 0,Y 509.842,Z 367.977,A -85,B 0,C 180,E1 -5454.625,E2 -5454.625} C_VEL
LIN {X 0,Y 509.862,Z 367.972,A -85,B 0,C 180,E1 -5457.482,E2 -5457.482} C_VEL
LIN {X 0,Y 509.879,Z 367.972,A -85,B 0,C 180,E1 -5460.27,E2 -5460.27} C_VEL
LIN {X 0,Y 509.886,Z 367.974,A -85,B 0,C 180,E1 -5462.946,E2 -5462.946} C_VEL
LIN {X 0,Y 509.901,Z 368.158,A -85,B 0,C 180,E1 -5465.462,E2 -5465.462} C_VEL
LIN {X 0,Y 511.533,Z 377.587,A -85,B 0,C 180,E1 -5467.141,E2 -5467.141} C_VEL
LIN {X 0,Y 511.033,Z 394.182,A -85,B 0,C 180,E1 -5469.892,E2 -5469.892} C_VEL
LIN {X 0,Y 510.531,Z 411.892,A -85,B 0,C 180,E1 -5472.786,E2 -5472.786} C_VEL
LIN {X 0,Y 510.266,Z 421.984,A -85,B 0,C 180,E1 -5474.42,E2 -5474.42} C_VEL
LIN {X 0,Y 512.254,Z 435.477,A -85,B 0,C 180,E1 -5474.678,E2 -5474.678} C_VEL
LIN {X 0,Y 511.713,Z 530.493,A -85,B 0,C 180,E1 -5476.043,E2 -5476.043} C_VEL
LIN {X 0,Y 511.458,Z 543.617,A -85,B 0,C 180,E1 -5476.391,E2 -5476.391} C_VEL
LIN {X 0,Y 511.158,Z 556.277,A -85,B 0,C 180,E1 -5476.889,E2 -5476.889} C_VEL
LIN {X 0,Y 510.88,Z 567.977,A -85,B 0,C 180,E1 -5477.516,E2 -5477.516} C_VEL
LIN {X 0,Y 510.558,Z 579.193,A -85,B 0,C 180,E1 -5478.286,E2 -5478.286} C_VEL
LIN {X 0,Y 510.242,Z 589.681,A -85,B 0,C 180,E1 -5479.184,E2 -5479.184} C_VEL
LIN {X 0,Y 509.941,Z 598.253,A -85,B 0,C 180,E1 -5480.081,E2 -5480.081} C_VEL
LIN {X 0,Y 509.694,Z 606.161,A -85,B 0,C 180,E1 -5481.077,E2 -5481.077} C_VEL
LIN {X 0,Y 509.487,Z 613.884,A -85,B 0,C 180,E1 -5482.272,E2 -5482.272} C_VEL
LIN {X 0,Y 509.321,Z 620.114,A -85,B 0,C 180,E1 -5483.471,E2 -5483.471} C_VEL
LIN {X 0,Y 509.244,Z 625.727,A -85,B 0,C 180,E1 -5484.854,E2 -5484.854} C_VEL
LIN {X 0,Y 509.245,Z 629.342,A -85,B 0,C 180,E1 -5486.044,E2 -5486.044} C_VEL
LIN {X 0,Y 509.2,Z 631.205,A -85,B 0,C 180,E1 -5486.836,E2 -5486.836} C_VEL
LIN {X 0,Y 509.189,Z 632.602,A -85,B 0,C 180,E1 -5487.628,E2 -5487.628} C_VEL
LIN {X 0,Y 509.073,Z 634.202,A -85,B 0,C 180,E1 -5489.21,E2 -5489.21} C_VEL
LIN {X 0,Y 509.065,Z 634.417,A -85,B 0,C 180,E1 -5490.001,E2 -5490.001} C_VEL
LIN {X 0,Y 509.112,Z 633.59,A -85,B 0,C 180,E1 -5491.583,E2 -5491.583} C_VEL
LIN {X 0,Y 509.189,Z 632.592,A -85,B 0,C 180,E1 -5492.374,E2 -5492.374} C_VEL
LIN {X 0,Y 509.201,Z 631.19,A -85,B 0,C 180,E1 -5493.166,E2 -5493.166} C_VEL
LIN {X 0,Y 509.205,Z 628.245,A -85,B 0,C 180,E1 -5494.355,E2 -5494.355} C_VEL
LIN {X 0,Y 509.3,Z 624.259,A -85,B 0,C 180,E1 -5495.544,E2 -5495.544} C_VEL
LIN {X 0,Y 509.402,Z 618.58,A -85,B 0,C 180,E1 -5496.845,E2 -5496.845} C_VEL
LIN {X 0,Y 509.552,Z 611.423,A -85,B 0,C 180,E1 -5498.128,E2 -5498.128} C_VEL
LIN {X 0,Y 509.776,Z 603.104,A -85,B 0,C 180,E1 -5499.323,E2 -5499.323} C_VEL
LIN {X 0,Y 510.015,Z 594.567,A -85,B 0,C 180,E1 -5500.321,E2 -5500.321} C_VEL
LIN {X 0,Y 510.386,Z 584.023,A -85,B 0,C 180,E1 -5501.317,E2 -5501.317} C_VEL
LIN {X 0,Y 510.672,Z 573.658,A -85,B 0,C 180,E1 -5502.111,E2 -5502.111} C_VEL
LIN {X 0,Y 511.027,Z 562.123,A -85,B 0,C 180,E1 -5502.813,E2 -5502.813} C_VEL
LIN {X 0,Y 511.311,Z 550.289,A -85,B 0,C 180,E1 -5503.362,E2 -5503.362} C_VEL
LIN {X 0,Y 511.558,Z 536.64,A -85,B 0,C 180,E1 -5503.811,E2 -5503.811} C_VEL
LIN {X 0,Y 511.792,Z 522.748,A -85,B 0,C 180,E1 -5504.083,E2 -5504.083} C_VEL
LIN {X 0,Y 512.161,Z 433.82,A -85,B 0,C 180,E1 -5505.346,E2 -5505.346} C_VEL
LIN {X 0,Y 510.258,Z 421.717,A -85,B 0,C 180,E1 -5505.596,E2 -5505.596} C_VEL
LIN {X 0,Y 510.758,Z 402.787,A -85,B 0,C 180,E1 -5508.659,E2 -5508.659} C_VEL
LIN {X 0,Y 511.303,Z 385.053,A -85,B 0,C 180,E1 -5511.574,E2 -5511.574} C_VEL
LIN {X 0,Y 511.491,Z 376.6,A -85,B 0,C 180,E1 -5512.986,E2 -5512.986} C_VEL
LIN {X 0,Y 509.882,Z 367.973,A -85,B 0,C 180,E1 -5514.533,E2 -5514.533} C_VEL
LIN {X 0,Y 509.891,Z 367.974,A -85,B 0,C 180,E1 -5517.056,E2 -5517.056} C_VEL
LIN {X 0,Y 509.863,Z 367.976,A -85,B 0,C 180,E1 -5519.752,E2 -5519.752} C_VEL
LIN {X 0,Y 509.879,Z 367.973,A -85,B 0,C 180,E1 -5522.775,E2 -5522.775} C_VEL
LIN {X 0,Y 509.834,Z 367.978,A -85,B 0,C 180,E1 -5525.579,E2 -5525.579} C_VEL
LIN {X 0,Y 509.856,Z 367.973,A -85,B 0,C 180,E1 -5528.338,E2 -5528.338} C_VEL
LIN {X 0,Y 509.861,Z 367.976,A -85,B 0,C 180,E1 -5531.426,E2 -5531.426} C_VEL
LIN {X 0,Y 509.863,Z 367.975,A -85,B 0,C 180,E1 -5534.668,E2 -5534.668} C_VEL
LIN {X 0,Y 509.861,Z 367.97,A -85,B 0,C 180,E1 -5538.104,E2 -5538.104} C_VEL
LIN {X 0,Y 509.851,Z 367.975,A -85,B 0,C 180,E1 -5540.648,E2 -5540.648} C_VEL
LIN {X 0,Y 509.83,Z 367.974,A -85,B 0,C 180,E1 -5543.647,E2 -5543.647} C_VEL
LIN {X 0,Y 509.864,Z 367.974,A -85,B 0,C 180,E1 -5546.539,E2 -5546.539} C_VEL
LIN {X 0,Y 509.851,Z 367.97,A -85,B 0,C 180,E1 -5549.335,E2 -5549.335} C_VEL
LIN {X 0,Y 509.894,Z 367.967,A -85,B 0,C 180,E1 -5552.054,E2 -5552.054} C_VEL
LIN {X 0,Y 509.846,Z 367.979,A -85,B 0,C 180,E1 -5554.702,E2 -5554.702} C_VEL
LIN {X 0,Y 509.832,Z 367.971,A -85,B 0,C 180,E1 -5557.458,E2 -5557.458} C_VEL
LIN {X 0,Y 509.922,Z 367.964,A -85,B 0,C 180,E1 -5559.845,E2 -5559.845} C_VEL
LIN {X 0,Y 509.887,Z 367.967,A -85,B 0,C 180,E1 -5563.175,E2 -5563.175} C_VEL
LIN {X 0,Y 509.869,Z 367.966,A -85,B 0,C 180,E1 -5565.634,E2 -5565.634} C_VEL
LIN {X 0,Y 509.919,Z 367.962,A -85,B 0,C 180,E1 -5568.875,E2 -5568.875} C_VEL
LIN {X 0,Y 509.957,Z 367.965,A -85,B 0,C 180,E1 -5572.079,E2 -5572.079} C_VEL
LIN {X 0,Y 509.987,Z 367.959,A -85,B 0,C 180,E1 -5574.464,E2 -5574.464} C_VEL
LIN {X 0,Y 510.061,Z 367.945,A -85,B 0,C 180,E1 -5577.631,E2 -5577.631} C_VEL
LIN {X 0,Y 510.069,Z 367.944,A -85,B 0,C 180,E1 -5580.79,E2 -5580.79} C_VEL
LIN {X 0,Y 509.96,Z 367.958,A -85,B 0,C 180,E1 -5583.16,E2 -5583.16} C_VEL
LIN {X 0,Y 509.985,Z 367.957,A -85,B 0,C 180,E1 -5586.33,E2 -5586.33} C_VEL
LIN {X 0,Y 509.92,Z 367.963,A -85,B 0,C 180,E1 -5588.72,E2 -5588.72} C_VEL
LIN {X 0,Y 509.911,Z 367.971,A -85,B 0,C 180,E1 -5591.932,E2 -5591.932} C_VEL
LIN {X 0,Y 509.9,Z 367.968,A -85,B 0,C 180,E1 -5595.242,E2 -5595.242} C_VEL
LIN {X 0,Y 509.888,Z 367.973,A -85,B 0,C 180,E1 -5597.998,E2 -5597.998} C_VEL
LIN {X 0,Y 509.857,Z 367.973,A -85,B 0,C 180,E1 -5601.002,E2 -5601.002} C_VEL
LIN {X 0,Y 509.829,Z 367.981,A -85,B 0,C 180,E1 -5603.564,E2 -5603.564} C_VEL
LIN {X 0,Y 509.917,Z 367.966,A -85,B 0,C 180,E1 -5606.378,E2 -5606.378} C_VEL
LIN {X 0,Y 509.882,Z 367.971,A -85,B 0,C 180,E1 -5608.844,E2 -5608.844} C_VEL
LIN {X 0,Y 509.855,Z 367.983,A -85,B 0,C 180,E1 -5611.009,E2 -5611.009} C_VEL
LIN {X 0,Y 510.828,Z 373.766,A -85,B 0,C 180,E1 -5612.217,E2 -5612.217} C_VEL
LIN {X 0,Y 510.449,Z 389.493,A -85,B 0,C 180,E1 -5615.329,E2 -5615.329} C_VEL
LIN {X 0,Y 510.301,Z 395.341,A -85,B 0,C 180,E1 -5616.474,E2 -5616.474} C_VEL
LIN {X 0,Y 512.301,Z 407.16,A -85,B 0,C 180,E1 -5616.719,E2 -5616.719} C_VEL
LIN {X 0,Y 511.711,Z 502.643,A -85,B 0,C 180,E1 -5618.096,E2 -5618.096} C_VEL
LIN {X 0,Y 511.511,Z 516.407,A -85,B 0,C 180,E1 -5618.47,E2 -5618.47} C_VEL
LIN {X 0,Y 510.761,Z 522.037,A -85,B 0,C 180,E1 -5618.657,E2 -5618.657} C_VEL
LIN {X 0,Y 507.7,Z 531.042,A -85,B 0,C 180,E1 -5618.981,E2 -5618.981} C_VEL
LIN {X 0,Y 504.63,Z 539.73,A -85,B 0,C 180,E1 -5619.391,E2 -5619.391} C_VEL
LIN {X 0,Y 503.864,Z 544.852,A -85,B 0,C 180,E1 -5619.71,E2 -5619.71} C_VEL
LIN {X 0,Y 503.519,Z 556.308,A -85,B 0,C 180,E1 -5620.601,E2 -5620.601} C_VEL
LIN {X 0,Y 503.119,Z 566.32,A -85,B 0,C 180,E1 -5621.569,E2 -5621.569} C_VEL
LIN {X 0,Y 502.85,Z 575.649,A -85,B 0,C 180,E1 -5622.692,E2 -5622.692} C_VEL
LIN {X 0,Y 502.542,Z 583.734,A -85,B 0,C 180,E1 -5623.898,E2 -5623.898} C_VEL
LIN {X 0,Y 502.368,Z 589.918,A -85,B 0,C 180,E1 -5625.039,E2 -5625.039} C_VEL
LIN {X 0,Y 502.26,Z 594.829,A -85,B 0,C 180,E1 -5626.16,E2 -5626.16} C_VEL
LIN {X 0,Y 502.173,Z 598.648,A -85,B 0,C 180,E1 -5627.252,E2 -5627.252} C_VEL
LIN {X 0,Y 502.127,Z 601.686,A -85,B 0,C 180,E1 -5628.377,E2 -5628.377} C_VEL
LIN {X 0,Y 501.995,Z 604.449,A -85,B 0,C 180,E1 -5629.908,E2 -5629.908} C_VEL
LIN {X 0,Y 501.996,Z 605.479,A -85,B 0,C 180,E1 -5630.949,E2 -5630.949} C_VEL
LIN {X 0,Y 501.978,Z 605.856,A -85,B 0,C 180,E1 -5631.973,E2 -5631.973} C_VEL
LIN {X 0,Y 501.948,Z 605.57,A -85,B 0,C 180,E1 -5632.981,E2 -5632.981} C_VEL
LIN {X 0,Y 501.998,Z 604.28,A -85,B 0,C 180,E1 -5634.293,E2 -5634.293} C_VEL
LIN {X 0,Y 502.105,Z 601.75,A -85,B 0,C 180,E1 -5635.673,E2 -5635.673} C_VEL
LIN {X 0,Y 502.173,Z 597.768,A -85,B 0,C 180,E1 -5637.11,E2 -5637.11} C_VEL
LIN {X 0,Y 502.319,Z 593.437,A -85,B 0,C 180,E1 -5638.267,E2 -5638.267} C_VEL
LIN {X 0,Y 502.444,Z 587.429,A -85,B 0,C 180,E1 -5639.531,E2 -5639.531} C_VEL
LIN {X 0,Y 502.655,Z 580.489,A -85,B 0,C 180,E1 -5640.7,E2 -5640.7} C_VEL
LIN {X 0,Y 502.953,Z 571.739,A -85,B 0,C 180,E1 -5641.891,E2 -5641.891} C_VEL
LIN {X 0,Y 503.295,Z 561.865,A -85,B 0,C 180,E1 -5642.972,E2 -5642.972} C_VEL
LIN {X 0,Y 503.684,Z 550.957,A -85,B 0,C 180,E1 -5643.925,E2 -5643.925} C_VEL
LIN {X 0,Y 504.012,Z 539.578,A -85,B 0,C 180,E1 -5644.719,E2 -5644.719} C_VEL
LIN {X 0,Y 504.385,Z 527.95,A -85,B 0,C 180,E1 -5645.345,E2 -5645.345} C_VEL
LIN {X 0,Y 504.603,Z 514.9,A -85,B 0,C 180,E1 -5645.863,E2 -5645.863} C_VEL
LIN {X 0,Y 504.843,Z 501.726,A -85,B 0,C 180,E1 -5646.208,E2 -5646.208} C_VEL
LIN {X 0,Y 505.303,Z 406.191,A -85,B 0,C 180,E1 -5647.604,E2 -5647.604} C_VEL
LIN {X 0,Y 503.276,Z 395.307,A -85,B 0,C 180,E1 -5647.849,E2 -5647.849} C_VEL
LIN {X 0,Y 503.712,Z 380.122,A -85,B 0,C 180,E1 -5650.859,E2 -5650.859} C_VEL
LIN {X 0,Y 503.747,Z 373.833,A -85,B 0,C 180,E1 -5652.125,E2 -5652.125} C_VEL
LIN {X 0,Y 502.871,Z 368.847,A -85,B 0,C 180,E1 -5653.194,E2 -5653.194} C_VEL
LIN {X 0,Y 502.837,Z 368.851,A -85,B 0,C 180,E1 -5656.254,E2 -5656.254} C_VEL
LIN {X 0,Y 502.883,Z 368.847,A -85,B 0,C 180,E1 -5658.716,E2 -5658.716} C_VEL
LIN {X 0,Y 502.907,Z 368.838,A -85,B 0,C 180,E1 -5661.966,E2 -5661.966} C_VEL
LIN {X 0,Y 502.932,Z 368.841,A -85,B 0,C 180,E1 -5664.385,E2 -5664.385} C_VEL
LIN {X 0,Y 503.03,Z 368.821,A -85,B 0,C 180,E1 -5667.597,E2 -5667.597} C_VEL
LIN {X 0,Y 503.032,Z 368.824,A -85,B 0,C 180,E1 -5669.999,E2 -5669.999} C_VEL
LIN {X 0,Y 503.029,Z 368.828,A -85,B 0,C 180,E1 -5672.401,E2 -5672.401} C_VEL
LIN {X 0,Y 502.941,Z 368.833,A -85,B 0,C 180,E1 -5675.612,E2 -5675.612} C_VEL
LIN {X 0,Y 502.904,Z 368.843,A -85,B 0,C 180,E1 -5678.032,E2 -5678.032} C_VEL
LIN {X 0,Y 502.88,Z 368.839,A -85,B 0,C 180,E1 -5681.282,E2 -5681.282} C_VEL
LIN {X 0,Y 502.847,Z 368.845,A -85,B 0,C 180,E1 -5684.57,E2 -5684.57} C_VEL
LIN {X 0,Y 502.863,Z 368.849,A -85,B 0,C 180,E1 -5687.906,E2 -5687.906} C_VEL
LIN {X 0,Y 502.829,Z 368.847,A -85,B 0,C 180,E1 -5690.535,E2 -5690.535} C_VEL
LIN {X 0,Y 502.789,Z 368.851,A -85,B 0,C 180,E1 -5693.039,E2 -5693.039} C_VEL
LIN {X 0,Y 502.821,Z 368.853,A -85,B 0,C 180,E1 -5695.675,E2 -5695.675} C_VEL
LIN {X 0,Y 502.84,Z 368.846,A -85,B 0,C 180,E1 -5698.371,E2 -5698.371} C_VEL
LIN {X 0,Y 502.795,Z 368.855,A -85,B 0,C 180,E1 -5701.498,E2 -5701.498} C_VEL
LIN {X 0,Y 502.804,Z 368.849,A -85,B 0,C 180,E1 -5704.443,E2 -5704.443} C_VEL
LIN {X 0,Y 502.778,Z 368.855,A -85,B 0,C 180,E1 -5707.177,E2 -5707.177} C_VEL
LIN {X 0,Y 502.817,Z 368.85,A -85,B 0,C 180,E1 -5710.011,E2 -5710.011} C_VEL
LIN {X 0,Y 502.798,Z 368.85,A -85,B 0,C 180,E1 -5712.198,E2 -5712.198} C_VEL
LIN {X 0,Y 502.795,Z 368.858,A -85,B 0,C 180,E1 -5715.467,E2 -5715.467} C_VEL
LIN {X 0,Y 502.862,Z 368.908,A -85,B 0,C 180,E1 -5717.342,E2 -5717.342} C_VEL
LIN {X 0,Y 503.587,Z 374.701,A -85,B 0,C 180,E1 -5718.463,E2 -5718.463} C_VEL
LIN {X 0,Y 503.314,Z 390.497,A -85,B 0,C 180,E1 -5721.437,E2 -5721.437} C_VEL
LIN {X 0,Y 503.257,Z 395.054,A -85,B 0,C 180,E1 -5722.275,E2 -5722.275} C_VEL
LIN {X 0,Y 505.374,Z 408.218,A -85,B 0,C 180,E1 -5722.545,E2 -5722.545} C_VEL
LIN {X 0,Y 504.726,Z 502.061,A -85,B 0,C 180,E1 -5723.942,E2 -5723.942} C_VEL
LIN {X 0,Y 504.515,Z 515.524,A -85,B 0,C 180,E1 -5724.299,E2 -5724.299} C_VEL
LIN {X 0,Y 504.244,Z 528.836,A -85,B 0,C 180,E1 -5724.844,E2 -5724.844} C_VEL
LIN {X 0,Y 503.935,Z 539.804,A -85,B 0,C 180,E1 -5725.443,E2 -5725.443} C_VEL
LIN {X 0,Y 503.619,Z 550.687,A -85,B 0,C 180,E1 -5726.198,E2 -5726.198} C_VEL
LIN {X 0,Y 503.256,Z 561.3,A -85,B 0,C 180,E1 -5727.119,E2 -5727.119} C_VEL
LIN {X 0,Y 502.937,Z 570.357,A -85,B 0,C 180,E1 -5728.086,E2 -5728.086} C_VEL
LIN {X 0,Y 502.708,Z 578.072,A -85,B 0,C 180,E1 -5729.084,E2 -5729.084} C_VEL
LIN {X 0,Y 502.458,Z 584.784,A -85,B 0,C 180,E1 -5730.133,E2 -5730.133} C_VEL
LIN {X 0,Y 502.332,Z 591.2,A -85,B 0,C 180,E1 -5731.368,E2 -5731.368} C_VEL
LIN {X 0,Y 502.195,Z 595.892,A -85,B 0,C 180,E1 -5732.495,E2 -5732.495} C_VEL
LIN {X 0,Y 502.143,Z 599.516,A -85,B 0,C 180,E1 -5733.601,E2 -5733.601} C_VEL
LIN {X 0,Y 502.102,Z 601.33,A -85,B 0,C 180,E1 -5734.284,E2 -5734.284} C_VEL
LIN {X 0,Y 502.009,Z 603.753,A -85,B 0,C 180,E1 -5735.499,E2 -5735.499} C_VEL
LIN {X 0,Y 501.981,Z 605.373,A -85,B 0,C 180,E1 -5736.92,E2 -5736.92} C_VEL
LIN {X 0,Y 502.001,Z 605.765,A -85,B 0,C 180,E1 -5737.79,E2 -5737.79} C_VEL
LIN {X 0,Y 501.98,Z 605.695,A -85,B 0,C 180,E1 -5738.653,E2 -5738.653} C_VEL
LIN {X 0,Y 502.028,Z 604.943,A -85,B 0,C 180,E1 -5739.705,E2 -5739.705} C_VEL
LIN {X 0,Y 502.063,Z 602.658,A -85,B 0,C 180,E1 -5741.218,E2 -5741.218} C_VEL
LIN {X 0,Y 502.138,Z 599.477,A -85,B 0,C 180,E1 -5742.517,E2 -5742.517} C_VEL
LIN {X 0,Y 502.182,Z 595.375,A -85,B 0,C 180,E1 -5743.746,E2 -5743.746} C_VEL
LIN {X 0,Y 502.385,Z 589.249,A -85,B 0,C 180,E1 -5745.141,E2 -5745.141} C_VEL
LIN {X 0,Y 502.591,Z 581.817,A -85,B 0,C 180,E1 -5746.454,E2 -5746.454} C_VEL
LIN {X 0,Y 502.881,Z 572.944,A -85,B 0,C 180,E1 -5747.694,E2 -5747.694} C_VEL
LIN {X 0,Y 503.141,Z 563.871,A -85,B 0,C 180,E1 -5748.723,E2 -5748.723} C_VEL
LIN {X 0,Y 503.542,Z 552.511,A -85,B 0,C 180,E1 -5749.749,E2 -5749.749} C_VEL
LIN {X 0,Y 503.951,Z 541.03,A -85,B 0,C 180,E1 -5750.569,E2 -5750.569} C_VEL
LIN {X 0,Y 504.223,Z 530.099,A -85,B 0,C 180,E1 -5751.18,E2 -5751.18} C_VEL
LIN {X 0,Y 504.476,Z 516.633,A -85,B 0,C 180,E1 -5751.744,E2 -5751.744} C_VEL
LIN {X 0,Y 504.726,Z 504.039,A -85,B 0,C 180,E1 -5752.096,E2 -5752.096} C_VEL
LIN {X 0,Y 504.91,Z 473.302,A -85,B 0,C 180,E1 -5752.577,E2 -5752.577} C_VEL
LIN {X 0,Y 505.305,Z 406.444,A -85,B 0,C 180,E1 -5753.574,E2 -5753.574} C_VEL
LIN {X 0,Y 503.254,Z 395.126,A -85,B 0,C 180,E1 -5753.837,E2 -5753.837} C_VEL
LIN {X 0,Y 503.509,Z 377.862,A -85,B 0,C 180,E1 -5757,E2 -5757} C_VEL
LIN {X 0,Y 503.323,Z 371.406,A -85,B 0,C 180,E1 -5758.2,E2 -5758.2} C_VEL
LIN {X 0,Y 502.914,Z 368.844,A -85,B 0,C 180,E1 -5758.699,E2 -5758.699} C_VEL
LIN {X 0,Y 503.026,Z 368.829,A -85,B 0,C 180,E1 -5760.8,E2 -5760.8} C_VEL
LIN {X 0,Y 502.894,Z 368.843,A -85,B 0,C 180,E1 -5763.204,E2 -5763.204} C_VEL
LIN {X 0,Y 502.918,Z 368.843,A -85,B 0,C 180,E1 -5766.419,E2 -5766.419} C_VEL
LIN {X 0,Y 502.867,Z 368.845,A -85,B 0,C 180,E1 -5768.843,E2 -5768.843} C_VEL
LIN {X 0,Y 502.882,Z 368.846,A -85,B 0,C 180,E1 -5772.101,E2 -5772.101} C_VEL
LIN {X 0,Y 502.837,Z 368.847,A -85,B 0,C 180,E1 -5775.4,E2 -5775.4} C_VEL
LIN {X 0,Y 502.835,Z 368.853,A -85,B 0,C 180,E1 -5778.123,E2 -5778.123} C_VEL
LIN {X 0,Y 502.791,Z 368.852,A -85,B 0,C 180,E1 -5781.311,E2 -5781.311} C_VEL
LIN {X 0,Y 502.81,Z 368.856,A -85,B 0,C 180,E1 -5783.913,E2 -5783.913} C_VEL
LIN {X 0,Y 502.871,Z 368.842,A -85,B 0,C 180,E1 -5786.566,E2 -5786.566} C_VEL
LIN {X 0,Y 502.83,Z 368.85,A -85,B 0,C 180,E1 -5789.288,E2 -5789.288} C_VEL
LIN {X 0,Y 502.78,Z 368.856,A -85,B 0,C 180,E1 -5792.085,E2 -5792.085} C_VEL
LIN {X 0,Y 502.802,Z 368.852,A -85,B 0,C 180,E1 -5794.966,E2 -5794.966} C_VEL
LIN {X 0,Y 502.786,Z 368.854,A -85,B 0,C 180,E1 -5797.955,E2 -5797.955} C_VEL
LIN {X 0,Y 502.813,Z 368.853,A -85,B 0,C 180,E1 -5801.067,E2 -5801.067} C_VEL
LIN {X 0,Y 502.783,Z 368.852,A -85,B 0,C 180,E1 -5804.34,E2 -5804.34} C_VEL
LIN {X 0,Y 502.779,Z 368.855,A -85,B 0,C 180,E1 -5806.771,E2 -5806.771} C_VEL
LIN {X 0,Y 502.813,Z 368.856,A -85,B 0,C 180,E1 -5809.006,E2 -5809.006} C_VEL
LIN {X 0,Y 502.789,Z 368.852,A -85,B 0,C 180,E1 -5812.047,E2 -5812.047} C_VEL
LIN {X 0,Y 502.806,Z 368.856,A -85,B 0,C 180,E1 -5815.036,E2 -5815.036} C_VEL
LIN {X 0,Y 502.785,Z 368.852,A -85,B 0,C 180,E1 -5817.917,E2 -5817.917} C_VEL
LIN {X 0,Y 502.837,Z 368.852,A -85,B 0,C 180,E1 -5820.714,E2 -5820.714} C_VEL
LIN {X 0,Y 502.879,Z 368.844,A -85,B 0,C 180,E1 -5823.436,E2 -5823.436} C_VEL
LIN {X 0,Y 502.837,Z 368.878,A -85,B 0,C 180,E1 -5825.247,E2 -5825.247} C_VEL
LIN {X 0,Y 504.612,Z 378.821,A -85,B 0,C 180,E1 -5827.049,E2 -5827.049} C_VEL
LIN {X 0,Y 504.058,Z 395.26,A -85,B 0,C 180,E1 -5829.814,E2 -5829.814} C_VEL
LIN {X 0,Y 503.531,Z 412.964,A -85,B 0,C 180,E1 -5832.748,E2 -5832.748} C_VEL
LIN {X 0,Y 503.259,Z 421.798,A -85,B 0,C 180,E1 -5834.198,E2 -5834.198} C_VEL
LIN {X 0,Y 505.424,Z 436.615,A -85,B 0,C 180,E1 -5834.485,E2 -5834.485} C_VEL
LIN {X 0,Y 504.822,Z 530.143,A -85,B 0,C 180,E1 -5835.849,E2 -5835.849} C_VEL
LIN {X 0,Y 504.568,Z 543.315,A -85,B 0,C 180,E1 -5836.201,E2 -5836.201} C_VEL
LIN {X 0,Y 504.229,Z 556,A -85,B 0,C 180,E1 -5836.705,E2 -5836.705} C_VEL
LIN {X 0,Y 503.961,Z 567.061,A -85,B 0,C 180,E1 -5837.299,E2 -5837.299} C_VEL
LIN {X 0,Y 503.586,Z 577.654,A -85,B 0,C 180,E1 -5838.02,E2 -5838.02} C_VEL
LIN {X 0,Y 503.28,Z 588.374,A -85,B 0,C 180,E1 -5838.931,E2 -5838.931} C_VEL
LIN {X 0,Y 502.918,Z 598.027,A -85,B 0,C 180,E1 -5839.941,E2 -5839.941} C_VEL
LIN {X 0,Y 502.657,Z 605.942,A -85,B 0,C 180,E1 -5840.951,E2 -5840.951} C_VEL
LIN {X 0,Y 502.408,Z 613.67,A -85,B 0,C 180,E1 -5842.162,E2 -5842.162} C_VEL
LIN {X 0,Y 502.226,Z 620.417,A -85,B 0,C 180,E1 -5843.492,E2 -5843.492} C_VEL
LIN {X 0,Y 502.176,Z 625.522,A -85,B 0,C 180,E1 -5844.782,E2 -5844.782} C_VEL
LIN {X 0,Y 502.138,Z 629.139,A -85,B 0,C 180,E1 -5845.988,E2 -5845.988} C_VEL
LIN {X 0,Y 502.12,Z 631.004,A -85,B 0,C 180,E1 -5846.792,E2 -5846.792} C_VEL
LIN {X 0,Y 502.091,Z 632.402,A -85,B 0,C 180,E1 -5847.594,E2 -5847.594} C_VEL
LIN {X 0,Y 501.99,Z 634.003,A -85,B 0,C 180,E1 -5849.199,E2 -5849.199} C_VEL
LIN {X 0,Y 501.98,Z 634.217,A -85,B 0,C 180,E1 -5850.001,E2 -5850.001} C_VEL
LIN {X 0,Y 502.036,Z 633.388,A -85,B 0,C 180,E1 -5851.605,E2 -5851.605} C_VEL
LIN {X 0,Y 502.091,Z 632.388,A -85,B 0,C 180,E1 -5852.408,E2 -5852.408} C_VEL
LIN {X 0,Y 502.12,Z 630.985,A -85,B 0,C 180,E1 -5853.21,E2 -5853.21} C_VEL
LIN {X 0,Y 502.103,Z 628.035,A -85,B 0,C 180,E1 -5854.416,E2 -5854.416} C_VEL
LIN {X 0,Y 502.217,Z 624.045,A -85,B 0,C 180,E1 -5855.623,E2 -5855.623} C_VEL
LIN {X 0,Y 502.333,Z 618.006,A -85,B 0,C 180,E1 -5857.013,E2 -5857.013} C_VEL
LIN {X 0,Y 502.483,Z 611.194,A -85,B 0,C 180,E1 -5858.243,E2 -5858.243} C_VEL
LIN {X 0,Y 502.733,Z 602.868,A -85,B 0,C 180,E1 -5859.455,E2 -5859.455} C_VEL
LIN {X 0,Y 502.994,Z 594.322,A -85,B 0,C 180,E1 -5860.466,E2 -5860.466} C_VEL
LIN {X 0,Y 503.407,Z 583.766,A -85,B 0,C 180,E1 -5861.476,E2 -5861.476} C_VEL
LIN {X 0,Y 503.685,Z 573.388,A -85,B 0,C 180,E1 -5862.281,E2 -5862.281} C_VEL
LIN {X 0,Y 504.069,Z 561.836,A -85,B 0,C 180,E1 -5862.993,E2 -5862.993} C_VEL
LIN {X 0,Y 504.39,Z 549.971,A -85,B 0,C 180,E1 -5863.549,E2 -5863.549} C_VEL
LIN {X 0,Y 504.643,Z 536.282,A -85,B 0,C 180,E1 -5864.004,E2 -5864.004} C_VEL
LIN {X 0,Y 504.889,Z 524.01,A -85,B 0,C 180,E1 -5864.254,E2 -5864.254} C_VEL
LIN {X 0,Y 505.292,Z 434.34,A -85,B 0,C 180,E1 -5865.55,E2 -5865.55} C_VEL
LIN {X 0,Y 503.254,Z 421.493,A -85,B 0,C 180,E1 -5865.819,E2 -5865.819} C_VEL
LIN {X 0,Y 503.765,Z 403.867,A -85,B 0,C 180,E1 -5868.717,E2 -5868.717} C_VEL
LIN {X 0,Y 504.337,Z 386.141,A -85,B 0,C 180,E1 -5871.672,E2 -5871.672} C_VEL
LIN {X 0,Y 504.48,Z 377.421,A -85,B 0,C 180,E1 -5873.153,E2 -5873.153} C_VEL
LIN {X 0,Y 502.85,Z 368.85,A -85,B 0,C 180,E1 -5874.747,E2 -5874.747} C_VEL
LIN {X 0,Y 502.84,Z 368.853,A -85,B 0,C 180,E1 -5877.467,E2 -5877.467} C_VEL
LIN {X 0,Y 502.815,Z 368.851,A -85,B 0,C 180,E1 -5880.212,E2 -5880.212} C_VEL
LIN {X 0,Y 502.837,Z 368.853,A -85,B 0,C 180,E1 -5883.032,E2 -5883.032} C_VEL
LIN {X 0,Y 502.78,Z 368.854,A -85,B 0,C 180,E1 -5885.952,E2 -5885.952} C_VEL
LIN {X 0,Y 502.808,Z 368.857,A -85,B 0,C 180,E1 -5888.976,E2 -5888.976} C_VEL
LIN {X 0,Y 502.801,Z 368.852,A -85,B 0,C 180,E1 -5892.14,E2 -5892.14} C_VEL
LIN {X 0,Y 502.807,Z 368.852,A -85,B 0,C 180,E1 -5895.469,E2 -5895.469} C_VEL
LIN {X 0,Y 502.825,Z 368.854,A -85,B 0,C 180,E1 -5898.934,E2 -5898.934} C_VEL
LIN {X 0,Y 502.798,Z 368.85,A -85,B 0,C 180,E1 -5902.046,E2 -5902.046} C_VEL
LIN {X 0,Y 502.804,Z 368.853,A -85,B 0,C 180,E1 -5905.034,E2 -5905.034} C_VEL
LIN {X 0,Y 502.789,Z 368.851,A -85,B 0,C 180,E1 -5907.916,E2 -5907.916} C_VEL
LIN {X 0,Y 502.829,Z 368.853,A -85,B 0,C 180,E1 -5910.712,E2 -5910.712} C_VEL
LIN {X 0,Y 502.868,Z 368.839,A -85,B 0,C 180,E1 -5913.439,E2 -5913.439} C_VEL
LIN {X 0,Y 502.781,Z 368.855,A -85,B 0,C 180,E1 -5916.086,E2 -5916.086} C_VEL
LIN {X 0,Y 502.789,Z 368.857,A -85,B 0,C 180,E1 -5918.689,E2 -5918.689} C_VEL
LIN {X 0,Y 502.834,Z 368.842,A -85,B 0,C 180,E1 -5921.248,E2 -5921.248} C_VEL
LIN {X 0,Y 502.827,Z 368.848,A -85,B 0,C 180,E1 -5923.767,E2 -5923.767} C_VEL
LIN {X 0,Y 502.836,Z 368.849,A -85,B 0,C 180,E1 -5926.255,E2 -5926.255} C_VEL
LIN {X 0,Y 502.883,Z 368.84,A -85,B 0,C 180,E1 -5928.717,E2 -5928.717} C_VEL
LIN {X 0,Y 502.907,Z 368.841,A -85,B 0,C 180,E1 -5931.967,E2 -5931.967} C_VEL
LIN {X 0,Y 502.943,Z 368.838,A -85,B 0,C 180,E1 -5934.387,E2 -5934.387} C_VEL
LIN {X 0,Y 503.03,Z 368.82,A -85,B 0,C 180,E1 -5937.598,E2 -5937.598} C_VEL
LIN {X 0,Y 503.033,Z 368.827,A -85,B 0,C 180,E1 -5940,E2 -5940} C_VEL
LIN {X 0,Y 503.03,Z 368.824,A -85,B 0,C 180,E1 -5942.402,E2 -5942.402} C_VEL
LIN {X 0,Y 502.944,Z 368.836,A -85,B 0,C 180,E1 -5945.614,E2 -5945.614} C_VEL
LIN {X 0,Y 502.908,Z 368.844,A -85,B 0,C 180,E1 -5948.033,E2 -5948.033} C_VEL
LIN {X 0,Y 502.883,Z 368.842,A -85,B 0,C 180,E1 -5951.283,E2 -5951.283} C_VEL
LIN {X 0,Y 502.851,Z 368.844,A -85,B 0,C 180,E1 -5954.571,E2 -5954.571} C_VEL
LIN {X 0,Y 502.861,Z 368.849,A -85,B 0,C 180,E1 -5957.907,E2 -5957.907} C_VEL
LIN {X 0,Y 502.835,Z 368.847,A -85,B 0,C 180,E1 -5960.536,E2 -5960.536} C_VEL
LIN {X 0,Y 502.794,Z 368.854,A -85,B 0,C 180,E1 -5963.041,E2 -5963.041} C_VEL
LIN {X 0,Y 502.828,Z 368.853,A -85,B 0,C 180,E1 -5965.676,E2 -5965.676} C_VEL
LIN {X 0,Y 502.846,Z 368.847,A -85,B 0,C 180,E1 -5968.373,E2 -5968.373} C_VEL
LIN {X 0,Y 502.816,Z 368.908,A -85,B 0,C 180,E1 -5970.85,E2 -5970.85} C_VEL
LIN {X 0,Y 503.885,Z 375.478,A -85,B 0,C 180,E1 -5972.242,E2 -5972.242} C_VEL
LIN {X 0,Y 503.442,Z 391.291,A -85,B 0,C 180,E1 -5975.404,E2 -5975.404} C_VEL
LIN {X 0,Y 503.313,Z 395.537,A -85,B 0,C 180,E1 -5976.247,E2 -5976.247} C_VEL
LIN {X 0,Y 505.452,Z 408.13,A -85,B 0,C 180,E1 -5976.517,E2 -5976.517} C_VEL
LIN {X 0,Y 504.831,Z 502.612,A -85,B 0,C 180,E1 -5977.9,E2 -5977.9} C_VEL
LIN {X 0,Y 504.611,Z 516.137,A -85,B 0,C 180,E1 -5978.268,E2 -5978.268} C_VEL
LIN {X 0,Y 504.348,Z 528.632,A -85,B 0,C 180,E1 -5978.774,E2 -5978.774} C_VEL
LIN {X 0,Y 504.018,Z 540.775,A -85,B 0,C 180,E1 -5979.444,E2 -5979.444} C_VEL
LIN {X 0,Y 503.864,Z 544.852,A -85,B 0,C 180,E1 -5979.71,E2 -5979.71} C_VEL
LIN {X 0,Y 503.087,Z 549.884,A -85,B 0,C 180,E1 -5980.059,E2 -5980.059} C_VEL
LIN {X 0,Y 499.942,Z 557.81,A -85,B 0,C 180,E1 -5980.643,E2 -5980.643} C_VEL
LIN {X 0,Y 496.794,Z 565.256,A -85,B 0,C 180,E1 -5981.302,E2 -5981.302} C_VEL
LIN {X 0,Y 496.015,Z 569.506,A -85,B 0,C 180,E1 -5981.763,E2 -5981.763} C_VEL
LIN {X 0,Y 495.746,Z 578.153,A -85,B 0,C 180,E1 -5982.881,E2 -5982.881} C_VEL
LIN {X 0,Y 495.467,Z 585.384,A -85,B 0,C 180,E1 -5984.031,E2 -5984.031} C_VEL
LIN {X 0,Y 495.274,Z 591.322,A -85,B 0,C 180,E1 -5985.195,E2 -5985.195} C_VEL
LIN {X 0,Y 495.15,Z 596.164,A -85,B 0,C 180,E1 -5986.376,E2 -5986.376} C_VEL
LIN {X 0,Y 495.069,Z 600.015,A -85,B 0,C 180,E1 -5987.578,E2 -5987.578} C_VEL
LIN {X 0,Y 494.999,Z 602.925,A -85,B 0,C 180,E1 -5988.807,E2 -5988.807} C_VEL
LIN {X 0,Y 494.904,Z 605.121,A -85,B 0,C 180,E1 -5990.279,E2 -5990.279} C_VEL
LIN {X 0,Y 494.91,Z 605.923,A -85,B 0,C 180,E1 -5991.355,E2 -5991.355} C_VEL
LIN {X 0,Y 494.885,Z 605.94,A -85,B 0,C 180,E1 -5992.681,E2 -5992.681} C_VEL
LIN {X 0,Y 494.901,Z 604.86,A -85,B 0,C 180,E1 -5994.042,E2 -5994.042} C_VEL
LIN {X 0,Y 495.007,Z 602.578,A -85,B 0,C 180,E1 -5995.434,E2 -5995.434} C_VEL
LIN {X 0,Y 495.092,Z 598.888,A -85,B 0,C 180,E1 -5996.88,E2 -5996.88} C_VEL
LIN {X 0,Y 495.253,Z 593.57,A -85,B 0,C 180,E1 -5998.37,E2 -5998.37} C_VEL
LIN {X 0,Y 495.391,Z 587.644,A -85,B 0,C 180,E1 -5999.633,E2 -5999.633} C_VEL
LIN {X 0,Y 495.661,Z 579.858,A -85,B 0,C 180,E1 -6000.945,E2 -6000.945} C_VEL
LIN {X 0,Y 495.963,Z 571.203,A -85,B 0,C 180,E1 -6002.119,E2 -6002.119} C_VEL
LIN {X 0,Y 496.33,Z 561.934,A -85,B 0,C 180,E1 -6003.136,E2 -6003.136} C_VEL
LIN {X 0,Y 496.72,Z 551.073,A -85,B 0,C 180,E1 -6004.096,E2 -6004.096} C_VEL
LIN {X 0,Y 497.081,Z 539.656,A -85,B 0,C 180,E1 -6004.902,E2 -6004.902} C_VEL
LIN {X 0,Y 497.456,Z 528.015,A -85,B 0,C 180,E1 -6005.535,E2 -6005.535} C_VEL
LIN {X 0,Y 497.717,Z 515.147,A -85,B 0,C 180,E1 -6006.052,E2 -6006.052} C_VEL
LIN {X 0,Y 497.962,Z 502.621,A -85,B 0,C 180,E1 -6006.389,E2 -6006.389} C_VEL
LIN {X 0,Y 498.602,Z 408.03,A -85,B 0,C 180,E1 -6007.793,E2 -6007.793} C_VEL
LIN {X 0,Y 496.291,Z 395.519,A -85,B 0,C 180,E1 -6008.068,E2 -6008.068} C_VEL
LIN {X 0,Y 496.772,Z 380.875,A -85,B 0,C 180,E1 -6011.01,E2 -6011.01} C_VEL
LIN {X 0,Y 496.697,Z 374.628,A -85,B 0,C 180,E1 -6012.288,E2 -6012.288} C_VEL
LIN {X 0,Y 495.825,Z 369.724,A -85,B 0,C 180,E1 -6013.372,E2 -6013.372} C_VEL
LIN {X 0,Y 495.8,Z 369.726,A -85,B 0,C 180,E1 -6016.055,E2 -6016.055} C_VEL
LIN {X 0,Y 495.858,Z 369.723,A -85,B 0,C 180,E1 -6018.554,E2 -6018.554} C_VEL
LIN {X 0,Y 495.879,Z 369.712,A -85,B 0,C 180,E1 -6021.851,E2 -6021.851} C_VEL
LIN {X 0,Y 495.843,Z 369.717,A -85,B 0,C 180,E1 -6025.12,E2 -6025.12} C_VEL
LIN {X 0,Y 495.998,Z 369.697,A -85,B 0,C 180,E1 -6027.563,E2 -6027.563} C_VEL
LIN {X 0,Y 496.009,Z 369.697,A -85,B 0,C 180,E1 -6030.811,E2 -6030.811} C_VEL
LIN {X 0,Y 495.845,Z 369.715,A -85,B 0,C 180,E1 -6033.249,E2 -6033.249} C_VEL
LIN {X 0,Y 495.883,Z 369.715,A -85,B 0,C 180,E1 -6036.509,E2 -6036.509} C_VEL
LIN {X 0,Y 495.842,Z 369.716,A -85,B 0,C 180,E1 -6038.969,E2 -6038.969} C_VEL
LIN {X 0,Y 495.831,Z 369.725,A -85,B 0,C 180,E1 -6042.034,E2 -6042.034} C_VEL
LIN {X 0,Y 495.825,Z 369.719,A -85,B 0,C 180,E1 -6045.45,E2 -6045.45} C_VEL
LIN {X 0,Y 495.808,Z 369.725,A -85,B 0,C 180,E1 -6048.246,E2 -6048.246} C_VEL
LIN {X 0,Y 495.774,Z 369.725,A -85,B 0,C 180,E1 -6050.755,E2 -6050.755} C_VEL
LIN {X 0,Y 495.743,Z 369.73,A -85,B 0,C 180,E1 -6053.386,E2 -6053.386} C_VEL
LIN {X 0,Y 495.822,Z 369.718,A -85,B 0,C 180,E1 -6056.748,E2 -6056.748} C_VEL
LIN {X 0,Y 495.78,Z 369.732,A -85,B 0,C 180,E1 -6059.744,E2 -6059.744} C_VEL
LIN {X 0,Y 495.767,Z 369.725,A -85,B 0,C 180,E1 -6062.593,E2 -6062.593} C_VEL
LIN {X 0,Y 495.755,Z 369.734,A -85,B 0,C 180,E1 -6065.535,E2 -6065.535} C_VEL
LIN {X 0,Y 495.772,Z 369.725,A -85,B 0,C 180,E1 -6068.769,E2 -6068.769} C_VEL
LIN {X 0,Y 495.773,Z 369.73,A -85,B 0,C 180,E1 -6071.778,E2 -6071.778} C_VEL
LIN {X 0,Y 495.743,Z 369.734,A -85,B 0,C 180,E1 -6075.138,E2 -6075.138} C_VEL
LIN {X 0,Y 495.804,Z 369.828,A -85,B 0,C 180,E1 -6077.23,E2 -6077.23} C_VEL
LIN {X 0,Y 496.574,Z 375.295,A -85,B 0,C 180,E1 -6078.303,E2 -6078.303} C_VEL
LIN {X 0,Y 496.357,Z 390.316,A -85,B 0,C 180,E1 -6081.144,E2 -6081.144} C_VEL
LIN {X 0,Y 496.253,Z 394.999,A -85,B 0,C 180,E1 -6082.029,E2 -6082.029} C_VEL
LIN {X 0,Y 498.532,Z 407.859,A -85,B 0,C 180,E1 -6082.321,E2 -6082.321} C_VEL
LIN {X 0,Y 497.819,Z 502.493,A -85,B 0,C 180,E1 -6083.759,E2 -6083.759} C_VEL
LIN {X 0,Y 497.609,Z 515.681,A -85,B 0,C 180,E1 -6084.117,E2 -6084.117} C_VEL
LIN {X 0,Y 497.303,Z 528.92,A -85,B 0,C 180,E1 -6084.665,E2 -6084.665} C_VEL
LIN {X 0,Y 496.967,Z 540.41,A -85,B 0,C 180,E1 -6085.303,E2 -6085.303} C_VEL
LIN {X 0,Y 496.591,Z 552.023,A -85,B 0,C 180,E1 -6086.134,E2 -6086.134} C_VEL
LIN {X 0,Y 496.23,Z 562.501,A -85,B 0,C 180,E1 -6087.078,E2 -6087.078} C_VEL
LIN {X 0,Y 495.885,Z 571.942,A -85,B 0,C 180,E1 -6088.126,E2 -6088.126} C_VEL
LIN {X 0,Y 495.613,Z 580.491,A -85,B 0,C 180,E1 -6089.303,E2 -6089.303} C_VEL
LIN {X 0,Y 495.351,Z 587.333,A -85,B 0,C 180,E1 -6090.46,E2 -6090.46} C_VEL
LIN {X 0,Y 495.186,Z 592.949,A -85,B 0,C 180,E1 -6091.632,E2 -6091.632} C_VEL
LIN {X 0,Y 495.088,Z 598.026,A -85,B 0,C 180,E1 -6092.983,E2 -6092.983} C_VEL
LIN {X 0,Y 495.008,Z 601.749,A -85,B 0,C 180,E1 -6094.34,E2 -6094.34} C_VEL
LIN {X 0,Y 494.91,Z 604.254,A -85,B 0,C 180,E1 -6095.681,E2 -6095.681} C_VEL
LIN {X 0,Y 494.901,Z 605.312,A -85,B 0,C 180,E1 -6096.57,E2 -6096.57} C_VEL
LIN {X 0,Y 494.91,Z 605.881,A -85,B 0,C 180,E1 -6097.454,E2 -6097.454} C_VEL
LIN {X 0,Y 494.879,Z 605.947,A -85,B 0,C 180,E1 -6098.331,E2 -6098.331} C_VEL
LIN {X 0,Y 494.922,Z 605.266,A -85,B 0,C 180,E1 -6099.585,E2 -6099.585} C_VEL
LIN {X 0,Y 494.967,Z 603.445,A -85,B 0,C 180,E1 -6100.939,E2 -6100.939} C_VEL
LIN {X 0,Y 495.038,Z 601.162,A -85,B 0,C 180,E1 -6102.02,E2 -6102.02} C_VEL
LIN {X 0,Y 495.114,Z 596.72,A -85,B 0,C 180,E1 -6103.507,E2 -6103.507} C_VEL
LIN {X 0,Y 495.252,Z 591.581,A -85,B 0,C 180,E1 -6104.784,E2 -6104.784} C_VEL
LIN {X 0,Y 495.458,Z 585.115,A -85,B 0,C 180,E1 -6106.046,E2 -6106.046} C_VEL
LIN {X 0,Y 495.704,Z 577.023,A -85,B 0,C 180,E1 -6107.305,E2 -6107.305} C_VEL
LIN {X 0,Y 496.027,Z 568.253,A -85,B 0,C 180,E1 -6108.409,E2 -6108.409} C_VEL
LIN {X 0,Y 496.359,Z 558.584,A -85,B 0,C 180,E1 -6109.393,E2 -6109.393} C_VEL
LIN {X 0,Y 496.753,Z 547.181,A -85,B 0,C 180,E1 -6110.328,E2 -6110.328} C_VEL
LIN {X 0,Y 497.103,Z 535.94,A -85,B 0,C 180,E1 -6111.053,E2 -6111.053} C_VEL
LIN {X 0,Y 497.427,Z 523.373,A -85,B 0,C 180,E1 -6111.671,E2 -6111.671} C_VEL
LIN {X 0,Y 497.683,Z 510.98,A -85,B 0,C 180,E1 -6112.112,E2 -6112.112} C_VEL
LIN {X 0,Y 497.854,Z 498.507,A -85,B 0,C 180,E1 -6112.395,E2 -6112.395} C_VEL
LIN {X 0,Y 498.499,Z 407.352,A -85,B 0,C 180,E1 -6113.778,E2 -6113.778} C_VEL
LIN {X 0,Y 496.273,Z 395.333,A -85,B 0,C 180,E1 -6114.056,E2 -6114.056} C_VEL
LIN {X 0,Y 496.563,Z 377.491,A -85,B 0,C 180,E1 -6117.363,E2 -6117.363} C_VEL
LIN {X 0,Y 496.236,Z 372.025,A -85,B 0,C 180,E1 -6118.377,E2 -6118.377} C_VEL
LIN {X 0,Y 495.888,Z 369.72,A -85,B 0,C 180,E1 -6118.833,E2 -6118.833} C_VEL
LIN {X 0,Y 495.996,Z 369.705,A -85,B 0,C 180,E1 -6120.812,E2 -6120.812} C_VEL
LIN {X 0,Y 495.838,Z 369.722,A -85,B 0,C 180,E1 -6123.25,E2 -6123.25} C_VEL
LIN {X 0,Y 495.869,Z 369.72,A -85,B 0,C 180,E1 -6126.51,E2 -6126.51} C_VEL
LIN {X 0,Y 495.835,Z 369.72,A -85,B 0,C 180,E1 -6128.97,E2 -6128.97} C_VEL
LIN {X 0,Y 495.84,Z 369.723,A -85,B 0,C 180,E1 -6132.275,E2 -6132.275} C_VEL
LIN {X 0,Y 495.797,Z 369.726,A -85,B 0,C 180,E1 -6135.624,E2 -6135.624} C_VEL
LIN {X 0,Y 495.795,Z 369.729,A -85,B 0,C 180,E1 -6138.248,E2 -6138.248} C_VEL
LIN {X 0,Y 495.767,Z 369.727,A -85,B 0,C 180,E1 -6140.757,E2 -6140.757} C_VEL
LIN {X 0,Y 495.764,Z 369.728,A -85,B 0,C 180,E1 -6143.386,E2 -6143.386} C_VEL
LIN {X 0,Y 495.793,Z 369.728,A -85,B 0,C 180,E1 -6146.068,E2 -6146.068} C_VEL
LIN {X 0,Y 495.771,Z 369.726,A -85,B 0,C 180,E1 -6148.815,E2 -6148.815} C_VEL
LIN {X 0,Y 495.751,Z 369.735,A -85,B 0,C 180,E1 -6151.727,E2 -6151.727} C_VEL
LIN {X 0,Y 495.768,Z 369.726,A -85,B 0,C 180,E1 -6154.696,E2 -6154.696} C_VEL
LIN {X 0,Y 495.724,Z 369.739,A -85,B 0,C 180,E1 -6157.562,E2 -6157.562} C_VEL
LIN {X 0,Y 495.759,Z 369.728,A -85,B 0,C 180,E1 -6160.701,E2 -6160.701} C_VEL
LIN {X 0,Y 495.728,Z 369.733,A -85,B 0,C 180,E1 -6163.697,E2 -6163.697} C_VEL
LIN {X 0,Y 495.727,Z 369.731,A -85,B 0,C 180,E1 -6166.306,E2 -6166.306} C_VEL
LIN {X 0,Y 495.761,Z 369.733,A -85,B 0,C 180,E1 -6169.301,E2 -6169.301} C_VEL
LIN {X 0,Y 495.727,Z 369.733,A -85,B 0,C 180,E1 -6172.44,E2 -6172.44} C_VEL
LIN {X 0,Y 495.781,Z 369.727,A -85,B 0,C 180,E1 -6175.459,E2 -6175.459} C_VEL
LIN {X 0,Y 495.756,Z 369.73,A -85,B 0,C 180,E1 -6178.365,E2 -6178.365} C_VEL
LIN {X 0,Y 495.788,Z 369.725,A -85,B 0,C 180,E1 -6181.507,E2 -6181.507} C_VEL
LIN {X 0,Y 495.798,Z 369.726,A -85,B 0,C 180,E1 -6183.934,E2 -6183.934} C_VEL
LIN {X 0,Y 495.82,Z 369.851,A -85,B 0,C 180,E1 -6185.074,E2 -6185.074} C_VEL
LIN {X 0,Y 497.665,Z 379.933,A -85,B 0,C 180,E1 -6186.93,E2 -6186.93} C_VEL
LIN {X 0,Y 497.1,Z 396.361,A -85,B 0,C 180,E1 -6189.735,E2 -6189.735} C_VEL
LIN {X 0,Y 496.531,Z 414.041,A -85,B 0,C 180,E1 -6192.709,E2 -6192.709} C_VEL
LIN {X 0,Y 496.262,Z 421.587,A -85,B 0,C 180,E1 -6193.966,E2 -6193.966} C_VEL
LIN {X 0,Y 498.595,Z 436.43,A -85,B 0,C 180,E1 -6194.267,E2 -6194.267} C_VEL
LIN {X 0,Y 497.958,Z 529.793,A -85,B 0,C 180,E1 -6195.65,E2 -6195.65} C_VEL
LIN {X 0,Y 497.655,Z 543.011,A -85,B 0,C 180,E1 -6196.006,E2 -6196.006} C_VEL
LIN {X 0,Y 497.315,Z 555.724,A -85,B 0,C 180,E1 -6196.517,E2 -6196.517} C_VEL
LIN {X 0,Y 496.986,Z 567.105,A -85,B 0,C 180,E1 -6197.137,E2 -6197.137} C_VEL
LIN {X 0,Y 496.558,Z 578.708,A -85,B 0,C 180,E1 -6197.951,E2 -6197.951} C_VEL
LIN {X 0,Y 496.25,Z 589.215,A -85,B 0,C 180,E1 -6198.876,E2 -6198.876} C_VEL
LIN {X 0,Y 495.875,Z 597.801,A -85,B 0,C 180,E1 -6199.797,E2 -6199.797} C_VEL
LIN {X 0,Y 495.618,Z 605.722,A -85,B 0,C 180,E1 -6200.822,E2 -6200.822} C_VEL
LIN {X 0,Y 495.357,Z 613.458,A -85,B 0,C 180,E1 -6202.05,E2 -6202.05} C_VEL
LIN {X 0,Y 495.252,Z 618.753,A -85,B 0,C 180,E1 -6203.073,E2 -6203.073} C_VEL
LIN {X 0,Y 495.134,Z 623.884,A -85,B 0,C 180,E1 -6204.299,E2 -6204.299} C_VEL
LIN {X 0,Y 495.008,Z 627.863,A -85,B 0,C 180,E1 -6205.522,E2 -6205.522} C_VEL
LIN {X 0,Y 495.041,Z 630.803,A -85,B 0,C 180,E1 -6206.746,E2 -6206.746} C_VEL
LIN {X 0,Y 494.997,Z 632.201,A -85,B 0,C 180,E1 -6207.56,E2 -6207.56} C_VEL
LIN {X 0,Y 494.962,Z 633.197,A -85,B 0,C 180,E1 -6208.374,E2 -6208.374} C_VEL
LIN {X 0,Y 494.898,Z 634.017,A -85,B 0,C 180,E1 -6210.001,E2 -6210.001} C_VEL
LIN {X 0,Y 494.962,Z 633.186,A -85,B 0,C 180,E1 -6211.628,E2 -6211.628} C_VEL
LIN {X 0,Y 494.998,Z 632.184,A -85,B 0,C 180,E1 -6212.442,E2 -6212.442} C_VEL
LIN {X 0,Y 495.042,Z 630.779,A -85,B 0,C 180,E1 -6213.256,E2 -6213.256} C_VEL
LIN {X 0,Y 495.009,Z 627.825,A -85,B 0,C 180,E1 -6214.48,E2 -6214.48} C_VEL
LIN {X 0,Y 495.135,Z 623.831,A -85,B 0,C 180,E1 -6215.703,E2 -6215.703} C_VEL
LIN {X 0,Y 495.258,Z 617.683,A -85,B 0,C 180,E1 -6217.134,E2 -6217.134} C_VEL
LIN {X 0,Y 495.43,Z 610.966,A -85,B 0,C 180,E1 -6218.362,E2 -6218.362} C_VEL
LIN {X 0,Y 495.693,Z 602.633,A -85,B 0,C 180,E1 -6219.591,E2 -6219.591} C_VEL
LIN {X 0,Y 495.992,Z 594.076,A -85,B 0,C 180,E1 -6220.616,E2 -6220.616} C_VEL
LIN {X 0,Y 496.43,Z 583.509,A -85,B 0,C 180,E1 -6221.64,E2 -6221.64} C_VEL
LIN {X 0,Y 496.756,Z 572.154,A -85,B 0,C 180,E1 -6222.525,E2 -6222.525} C_VEL
LIN {X 0,Y 497.136,Z 561.548,A -85,B 0,C 180,E1 -6223.178,E2 -6223.178} C_VEL
LIN {X 0,Y 497.456,Z 549.653,A -85,B 0,C 180,E1 -6223.741,E2 -6223.741} C_VEL
LIN {X 0,Y 497.768,Z 535.926,A -85,B 0,C 180,E1 -6224.202,E2 -6224.202} C_VEL
LIN {X 0,Y 498.027,Z 523.553,A -85,B 0,C 180,E1 -6224.455,E2 -6224.455} C_VEL
LIN {X 0,Y 498.4,Z 434.748,A -85,B 0,C 180,E1 -6225.761,E2 -6225.761} C_VEL
LIN {X 0,Y 496.248,Z 421.344,A -85,B 0,C 180,E1 -6226.038,E2 -6226.038} C_VEL
LIN {X 0,Y 496.798,Z 403.673,A -85,B 0,C 180,E1 -6228.989,E2 -6228.989} C_VEL
LIN {X 0,Y 497.377,Z 387.229,A -85,B 0,C 180,E1 -6231.773,E2 -6231.773} C_VEL
LIN {X 0,Y 497.487,Z 378.391,A -85,B 0,C 180,E1 -6233.302,E2 -6233.302} C_VEL
LIN {X 0,Y 495.802,Z 369.729,A -85,B 0,C 180,E1 -6234.932,E2 -6234.932} C_VEL
LIN {X 0,Y 495.787,Z 369.73,A -85,B 0,C 180,E1 -6237.892,E2 -6237.892} C_VEL
LIN {X 0,Y 495.757,Z 369.732,A -85,B 0,C 180,E1 -6240.688,E2 -6240.688} C_VEL
LIN {X 0,Y 495.766,Z 369.731,A -85,B 0,C 180,E1 -6243.565,E2 -6243.565} C_VEL
LIN {X 0,Y 495.734,Z 369.733,A -85,B 0,C 180,E1 -6246.544,E2 -6246.544} C_VEL
LIN {X 0,Y 495.763,Z 369.731,A -85,B 0,C 180,E1 -6249.638,E2 -6249.638} C_VEL
LIN {X 0,Y 495.743,Z 369.733,A -85,B 0,C 180,E1 -6252.507,E2 -6252.507} C_VEL
LIN {X 0,Y 495.755,Z 369.735,A -85,B 0,C 180,E1 -6255.14,E2 -6255.14} C_VEL
LIN {X 0,Y 495.761,Z 369.727,A -85,B 0,C 180,E1 -6258.219,E2 -6258.219} C_VEL
LIN {X 0,Y 495.755,Z 369.729,A -85,B 0,C 180,E1 -6261.409,E2 -6261.409} C_VEL
LIN {X 0,Y 495.753,Z 369.731,A -85,B 0,C 180,E1 -6264.463,E2 -6264.463} C_VEL
LIN {X 0,Y 495.773,Z 369.726,A -85,B 0,C 180,E1 -6267.406,E2 -6267.406} C_VEL
LIN {X 0,Y 495.771,Z 369.725,A -85,B 0,C 180,E1 -6270.254,E2 -6270.254} C_VEL
LIN {X 0,Y 495.829,Z 369.717,A -85,B 0,C 180,E1 -6273.251,E2 -6273.251} C_VEL
LIN {X 0,Y 495.748,Z 369.732,A -85,B 0,C 180,E1 -6276.613,E2 -6276.613} C_VEL
LIN {X 0,Y 495.784,Z 369.724,A -85,B 0,C 180,E1 -6279.324,E2 -6279.324} C_VEL
LIN {X 0,Y 495.798,Z 369.72,A -85,B 0,C 180,E1 -6281.829,E2 -6281.829} C_VEL
LIN {X 0,Y 495.83,Z 369.721,A -85,B 0,C 180,E1 -6284.549,E2 -6284.549} C_VEL
LIN {X 0,Y 495.834,Z 369.722,A -85,B 0,C 180,E1 -6287.965,E2 -6287.965} C_VEL
LIN {X 0,Y 495.847,Z 369.717,A -85,B 0,C 180,E1 -6291.03,E2 -6291.03} C_VEL
LIN {X 0,Y 495.886,Z 369.709,A -85,B 0,C 180,E1 -6293.49,E2 -6293.49} C_VEL
LIN {X 0,Y 495.847,Z 369.714,A -85,B 0,C 180,E1 -6296.75,E2 -6296.75} C_VEL
LIN {X 0,Y 495.876,Z 369.717,A -85,B 0,C 180,E1 -6298.376,E2 -6298.376} C_VEL
LIN {X 0,Y 495.989,Z 369.698,A -85,B 0,C 180,E1 -6300.812,E2 -6300.812} C_VEL
LIN {X 0,Y 495.999,Z 369.7,A -85,B 0,C 180,E1 -6302.436,E2 -6302.436} C_VEL
LIN {X 0,Y 495.901,Z 369.715,A -85,B 0,C 180,E1 -6305.694,E2 -6305.694} C_VEL
LIN {X 0,Y 495.879,Z 369.718,A -85,B 0,C 180,E1 -6308.148,E2 -6308.148} C_VEL
LIN {X 0,Y 495.858,Z 369.719,A -85,B 0,C 180,E1 -6311.445,E2 -6311.445} C_VEL
LIN {X 0,Y 495.796,Z 369.723,A -85,B 0,C 180,E1 -6314.783,E2 -6314.783} C_VEL
LIN {X 0,Y 495.788,Z 369.728,A -85,B 0,C 180,E1 -6317.319,E2 -6317.319} C_VEL
LIN {X 0,Y 495.777,Z 369.731,A -85,B 0,C 180,E1 -6319.89,E2 -6319.89} C_VEL
LIN {X 0,Y 495.765,Z 369.728,A -85,B 0,C 180,E1 -6322.86,E2 -6322.86} C_VEL
LIN {X 0,Y 495.787,Z 369.728,A -85,B 0,C 180,E1 -6326.068,E2 -6326.068} C_VEL
LIN {X 0,Y 495.778,Z 369.729,A -85,B 0,C 180,E1 -6328.815,E2 -6328.815} C_VEL
LIN {X 0,Y 495.788,Z 369.828,A -85,B 0,C 180,E1 -6330.685,E2 -6330.685} C_VEL
LIN {X 0,Y 496.927,Z 376.599,A -85,B 0,C 180,E1 -6332.144,E2 -6332.144} C_VEL
LIN {X 0,Y 496.492,Z 391.218,A -85,B 0,C 180,E1 -6335.107,E2 -6335.107} C_VEL
LIN {X 0,Y 496.362,Z 395.8,A -85,B 0,C 180,E1 -6336.027,E2 -6336.027} C_VEL
LIN {X 0,Y 498.64,Z 409.153,A -85,B 0,C 180,E1 -6336.312,E2 -6336.312} C_VEL
LIN {X 0,Y 497.967,Z 503.02,A -85,B 0,C 180,E1 -6337.71,E2 -6337.71} C_VEL
LIN {X 0,Y 497.715,Z 516.495,A -85,B 0,C 180,E1 -6338.083,E2 -6338.083} C_VEL
LIN {X 0,Y 497.455,Z 528.872,A -85,B 0,C 180,E1 -6338.592,E2 -6338.592} C_VEL
LIN {X 0,Y 497.081,Z 541.243,A -85,B 0,C 180,E1 -6339.287,E2 -6339.287} C_VEL
LIN {X 0,Y 496.712,Z 551.517,A -85,B 0,C 180,E1 -6340.023,E2 -6340.023} C_VEL
LIN {X 0,Y 496.331,Z 562.295,A -85,B 0,C 180,E1 -6340.982,E2 -6340.982} C_VEL
LIN {X 0,Y 496.015,Z 569.506,A -85,B 0,C 180,E1 -6341.763,E2 -6341.763} C_VEL
LIN {X 0,Y 495.274,Z 573.6,A -85,B 0,C 180,E1 -6342.248,E2 -6342.248} C_VEL
LIN {X 0,Y 492.249,Z 579.952,A -85,B 0,C 180,E1 -6343.06,E2 -6343.06} C_VEL
LIN {X 0,Y 489.16,Z 585.668,A -85,B 0,C 180,E1 -6343.938,E2 -6343.938} C_VEL
LIN {X 0,Y 488.333,Z 588.767,A -85,B 0,C 180,E1 -6344.521,E2 -6344.521} C_VEL
LIN {X 0,Y 488.162,Z 593.802,A -85,B 0,C 180,E1 -6345.626,E2 -6345.626} C_VEL
LIN {X 0,Y 488.039,Z 598.094,A -85,B 0,C 180,E1 -6346.802,E2 -6346.802} C_VEL
LIN {X 0,Y 487.957,Z 601.339,A -85,B 0,C 180,E1 -6347.952,E2 -6347.952} C_VEL
LIN {X 0,Y 487.816,Z 604.496,A -85,B 0,C 180,E1 -6349.584,E2 -6349.584} C_VEL
LIN {X 0,Y 487.799,Z 605.973,A -85,B 0,C 180,E1 -6351.079,E2 -6351.079} C_VEL
LIN {X 0,Y 487.801,Z 606.109,A -85,B 0,C 180,E1 -6352.762,E2 -6352.762} C_VEL
LIN {X 0,Y 487.781,Z 605.349,A -85,B 0,C 180,E1 -6353.79,E2 -6353.79} C_VEL
LIN {X 0,Y 487.883,Z 603.334,A -85,B 0,C 180,E1 -6355.195,E2 -6355.195} C_VEL
LIN {X 0,Y 487.979,Z 599.968,A -85,B 0,C 180,E1 -6356.651,E2 -6356.651} C_VEL
LIN {X 0,Y 488.155,Z 594.97,A -85,B 0,C 180,E1 -6358.15,E2 -6358.15} C_VEL
LIN {X 0,Y 488.3,Z 588.982,A -85,B 0,C 180,E1 -6359.512,E2 -6359.512} C_VEL
LIN {X 0,Y 488.555,Z 582.314,A -85,B 0,C 180,E1 -6360.718,E2 -6360.718} C_VEL
LIN {X 0,Y 488.884,Z 574.114,A -85,B 0,C 180,E1 -6361.913,E2 -6361.913} C_VEL
LIN {X 0,Y 489.248,Z 564.546,A -85,B 0,C 180,E1 -6363.04,E2 -6363.04} C_VEL
LIN {X 0,Y 489.717,Z 554.012,A -85,B 0,C 180,E1 -6364.041,E2 -6364.041} C_VEL
LIN {X 0,Y 490.062,Z 543.25,A -85,B 0,C 180,E1 -6364.858,E2 -6364.858} C_VEL
LIN {X 0,Y 490.451,Z 531.502,A -85,B 0,C 180,E1 -6365.557,E2 -6365.557} C_VEL
LIN {X 0,Y 490.754,Z 519.983,A -85,B 0,C 180,E1 -6366.079,E2 -6366.079} C_VEL
LIN {X 0,Y 491.051,Z 507.264,A -85,B 0,C 180,E1 -6366.486,E2 -6366.486} C_VEL
LIN {X 0,Y 491.188,Z 491.84,A -85,B 0,C 180,E1 -6366.772,E2 -6366.772} C_VEL
LIN {X 0,Y 491.697,Z 408.229,A -85,B 0,C 180,E1 -6368.018,E2 -6368.018} C_VEL
LIN {X 0,Y 489.333,Z 395.726,A -85,B 0,C 180,E1 -6368.294,E2 -6368.294} C_VEL
LIN {X 0,Y 489.823,Z 381.169,A -85,B 0,C 180,E1 -6371.258,E2 -6371.258} C_VEL
LIN {X 0,Y 489.907,Z 377.399,A -85,B 0,C 180,E1 -6372.034,E2 -6372.034} C_VEL
LIN {X 0,Y 488.786,Z 370.601,A -85,B 0,C 180,E1 -6373.528,E2 -6373.528} C_VEL
LIN {X 0,Y 488.738,Z 370.61,A -85,B 0,C 180,E1 -6376.697,E2 -6376.697} C_VEL
LIN {X 0,Y 488.745,Z 370.601,A -85,B 0,C 180,E1 -6379.225,E2 -6379.225} C_VEL
LIN {X 0,Y 488.823,Z 370.591,A -85,B 0,C 180,E1 -6381.733,E2 -6381.733} C_VEL
LIN {X 0,Y 488.812,Z 370.593,A -85,B 0,C 180,E1 -6385.05,E2 -6385.05} C_VEL
LIN {X 0,Y 488.966,Z 370.573,A -85,B 0,C 180,E1 -6387.528,E2 -6387.528} C_VEL
LIN {X 0,Y 488.958,Z 370.576,A -85,B 0,C 180,E1 -6390.822,E2 -6390.822} C_VEL
LIN {X 0,Y 488.965,Z 370.578,A -85,B 0,C 180,E1 -6392.47,E2 -6392.47} C_VEL
LIN {X 0,Y 488.858,Z 370.589,A -85,B 0,C 180,E1 -6395.775,E2 -6395.775} C_VEL
LIN {X 0,Y 488.819,Z 370.598,A -85,B 0,C 180,E1 -6398.265,E2 -6398.265} C_VEL
LIN {X 0,Y 488.808,Z 370.594,A -85,B 0,C 180,E1 -6401.611,E2 -6401.611} C_VEL
LIN {X 0,Y 488.764,Z 370.598,A -85,B 0,C 180,E1 -6404.999,E2 -6404.999} C_VEL
LIN {X 0,Y 488.756,Z 370.601,A -85,B 0,C 180,E1 -6408.441,E2 -6408.441} C_VEL
LIN {X 0,Y 488.707,Z 370.605,A -85,B 0,C 180,E1 -6411.069,E2 -6411.069} C_VEL
LIN {X 0,Y 488.677,Z 370.615,A -85,B 0,C 180,E1 -6413.745,E2 -6413.745} C_VEL
LIN {X 0,Y 488.791,Z 370.594,A -85,B 0,C 180,E1 -6416.942,E2 -6416.942} C_VEL
LIN {X 0,Y 488.717,Z 370.605,A -85,B 0,C 180,E1 -6420.363,E2 -6420.363} C_VEL
LIN {X 0,Y 488.733,Z 370.607,A -85,B 0,C 180,E1 -6423.483,E2 -6423.483} C_VEL
LIN {X 0,Y 488.686,Z 370.608,A -85,B 0,C 180,E1 -6426.354,E2 -6426.354} C_VEL
LIN {X 0,Y 488.741,Z 370.604,A -85,B 0,C 180,E1 -6429.249,E2 -6429.249} C_VEL
LIN {X 0,Y 488.69,Z 370.607,A -85,B 0,C 180,E1 -6432.524,E2 -6432.524} C_VEL
LIN {X 0,Y 488.706,Z 370.612,A -85,B 0,C 180,E1 -6435.198,E2 -6435.198} C_VEL
LIN {X 0,Y 488.773,Z 370.661,A -85,B 0,C 180,E1 -6437.107,E2 -6437.107} C_VEL
LIN {X 0,Y 489.616,Z 376.621,A -85,B 0,C 180,E1 -6438.278,E2 -6438.278} C_VEL
LIN {X 0,Y 489.318,Z 392.656,A -85,B 0,C 180,E1 -6441.334,E2 -6441.334} C_VEL
LIN {X 0,Y 489.279,Z 395.463,A -85,B 0,C 180,E1 -6441.822,E2 -6441.822} C_VEL
LIN {X 0,Y 491.691,Z 409.411,A -85,B 0,C 180,E1 -6442.123,E2 -6442.123} C_VEL
LIN {X 0,Y 490.944,Z 502.86,A -85,B 0,C 180,E1 -6443.572,E2 -6443.572} C_VEL
LIN {X 0,Y 490.722,Z 515.396,A -85,B 0,C 180,E1 -6443.916,E2 -6443.916} C_VEL
LIN {X 0,Y 490.427,Z 527.529,A -85,B 0,C 180,E1 -6444.409,E2 -6444.409} C_VEL
LIN {X 0,Y 490.038,Z 540.357,A -85,B 0,C 180,E1 -6445.119,E2 -6445.119} C_VEL
LIN {X 0,Y 489.636,Z 552,A -85,B 0,C 180,E1 -6445.959,E2 -6445.959} C_VEL
LIN {X 0,Y 489.225,Z 562.501,A -85,B 0,C 180,E1 -6446.914,E2 -6446.914} C_VEL
LIN {X 0,Y 488.849,Z 572.3,A -85,B 0,C 180,E1 -6448.016,E2 -6448.016} C_VEL
LIN {X 0,Y 488.603,Z 579.977,A -85,B 0,C 180,E1 -6449.078,E2 -6449.078} C_VEL
LIN {X 0,Y 488.303,Z 588.066,A -85,B 0,C 180,E1 -6450.465,E2 -6450.465} C_VEL
LIN {X 0,Y 488.101,Z 593.48,A -85,B 0,C 180,E1 -6451.63,E2 -6451.63} C_VEL
LIN {X 0,Y 488.002,Z 598.274,A -85,B 0,C 180,E1 -6452.937,E2 -6452.937} C_VEL
LIN {X 0,Y 487.922,Z 602.168,A -85,B 0,C 180,E1 -6454.398,E2 -6454.398} C_VEL
LIN {X 0,Y 487.848,Z 603.926,A -85,B 0,C 180,E1 -6455.305,E2 -6455.305} C_VEL
LIN {X 0,Y 487.797,Z 605.162,A -85,B 0,C 180,E1 -6456.208,E2 -6456.208} C_VEL
LIN {X 0,Y 487.798,Z 605.96,A -85,B 0,C 180,E1 -6457.229,E2 -6457.229} C_VEL
LIN {X 0,Y 487.801,Z 606.172,A -85,B 0,C 180,E1 -6458.001,E2 -6458.001} C_VEL
LIN {X 0,Y 487.843,Z 605.595,A -85,B 0,C 180,E1 -6459.452,E2 -6459.452} C_VEL
LIN {X 0,Y 487.848,Z 604.189,A -85,B 0,C 180,E1 -6460.65,E2 -6460.65} C_VEL
LIN {X 0,Y 487.95,Z 601.749,A -85,B 0,C 180,E1 -6461.911,E2 -6461.911} C_VEL
LIN {X 0,Y 487.996,Z 597.987,A -85,B 0,C 180,E1 -6463.259,E2 -6463.259} C_VEL
LIN {X 0,Y 488.169,Z 592.532,A -85,B 0,C 180,E1 -6464.698,E2 -6464.698} C_VEL
LIN {X 0,Y 488.41,Z 585.874,A -85,B 0,C 180,E1 -6466.053,E2 -6466.053} C_VEL
LIN {X 0,Y 488.659,Z 577.897,A -85,B 0,C 180,E1 -6467.33,E2 -6467.33} C_VEL
LIN {X 0,Y 488.967,Z 569.758,A -85,B 0,C 180,E1 -6468.391,E2 -6468.391} C_VEL
LIN {X 0,Y 489.357,Z 559.818,A -85,B 0,C 180,E1 -6469.449,E2 -6469.449} C_VEL
LIN {X 0,Y 489.735,Z 548.638,A -85,B 0,C 180,E1 -6470.397,E2 -6470.397} C_VEL
LIN {X 0,Y 490.159,Z 536.558,A -85,B 0,C 180,E1 -6471.203,E2 -6471.203} C_VEL
LIN {X 0,Y 490.517,Z 524.442,A -85,B 0,C 180,E1 -6471.814,E2 -6471.814} C_VEL
LIN {X 0,Y 490.772,Z 511.68,A -85,B 0,C 180,E1 -6472.284,E2 -6472.284} C_VEL
LIN {X 0,Y 490.965,Z 498.146,A -85,B 0,C 180,E1 -6472.598,E2 -6472.598} C_VEL
LIN {X 0,Y 491.609,Z 407.919,A -85,B 0,C 180,E1 -6473.999,E2 -6473.999} C_VEL
LIN {X 0,Y 489.29,Z 395.425,A -85,B 0,C 180,E1 -6474.307,E2 -6474.307} C_VEL
LIN {X 0,Y 489.587,Z 378.147,A -85,B 0,C 180,E1 -6477.532,E2 -6477.532} C_VEL
LIN {X 0,Y 489.17,Z 372.642,A -85,B 0,C 180,E1 -6478.559,E2 -6478.559} C_VEL
LIN {X 0,Y 488.885,Z 370.591,A -85,B 0,C 180,E1 -6478.97,E2 -6478.97} C_VEL
LIN {X 0,Y 488.967,Z 370.58,A -85,B 0,C 180,E1 -6480.823,E2 -6480.823} C_VEL
LIN {X 0,Y 488.952,Z 370.584,A -85,B 0,C 180,E1 -6482.471,E2 -6482.471} C_VEL
LIN {X 0,Y 488.846,Z 370.592,A -85,B 0,C 180,E1 -6485.776,E2 -6485.776} C_VEL
